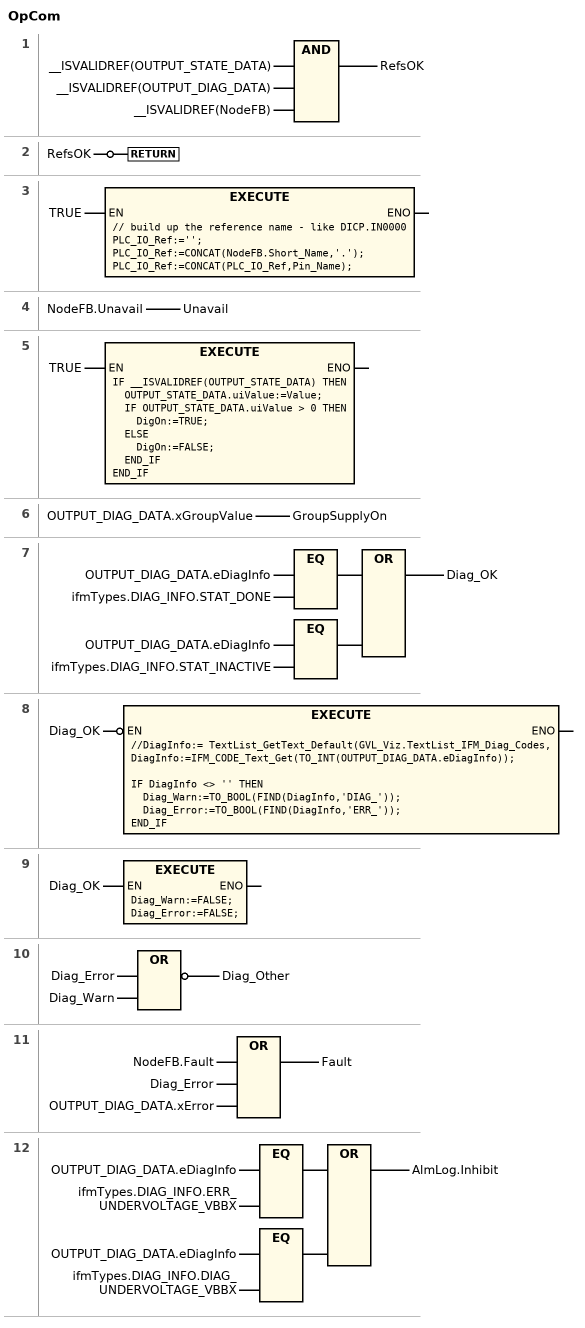
// NETWORK 1
RefsOK := (__ISVALIDREF(OUTPUT_STATE_DATA)) AND (__ISVALIDREF(OUTPUT_DIAG_DATA)) AND (__ISVALIDREF(NodeFB));

// NETWORK 2
IF NOT RefsOK THEN RETURN; END_IF

// NETWORK 3
// build up the reference name - like DICP.IN0000
PLC_IO_Ref:='';
PLC_IO_Ref:=CONCAT(NodeFB.Short_Name,'.');
PLC_IO_Ref:=CONCAT(PLC_IO_Ref,Pin_Name);

// NETWORK 4
Unavail := NodeFB.Unavail;

// NETWORK 5
IF __ISVALIDREF(OUTPUT_STATE_DATA) THEN
	OUTPUT_STATE_DATA.uiValue:=Value;
	IF OUTPUT_STATE_DATA.uiValue > 0 THEN
		DigOn:=TRUE;
	ELSE
		DigOn:=FALSE;
	END_IF
END_IF

// NETWORK 6
GroupSupplyOn := OUTPUT_DIAG_DATA.xGroupValue;

// NETWORK 7
Diag_OK := OUTPUT_DIAG_DATA.eDiagInfo = ifmTypes.DIAG_INFO.STAT_DONE OR OUTPUT_DIAG_DATA.eDiagInfo = ifmTypes.DIAG_INFO.STAT_INACTIVE;

// NETWORK 8
IF NOT Diag_OK THEN
    //DiagInfo:= TextList_GetText_Default(GVL_Viz.TextList_IFM_Diag_Codes,TO_STRING(OUTPUT_DIAG_DATA.eDiagInfo));
    DiagInfo:=IFM_CODE_Text_Get(TO_INT(OUTPUT_DIAG_DATA.eDiagInfo));
    
    IF DiagInfo <> '' THEN
    	Diag_Warn:=TO_BOOL(FIND(DiagInfo,'DIAG_'));	
    	Diag_Error:=TO_BOOL(FIND(DiagInfo,'ERR_'));	
    END_IF
END_IF

// NETWORK 9
IF Diag_OK THEN
    Diag_Warn:=FALSE;
    Diag_Error:=FALSE;
END_IF

// NETWORK 10
Diag_Other := NOT (Diag_Error OR Diag_Warn);

// NETWORK 11
Fault := NodeFB.Fault OR Diag_Error OR OUTPUT_DIAG_DATA.xError;

// NETWORK 12
AlmLog.Inhibit := OUTPUT_DIAG_DATA.eDiagInfo = ifmTypes.DIAG_INFO.ERR_UNDERVOLTAGE_VBBX OR OUTPUT_DIAG_DATA.eDiagInfo = ifmTypes.DIAG_INFO.DIAG_UNDERVOLTAGE_VBBX;

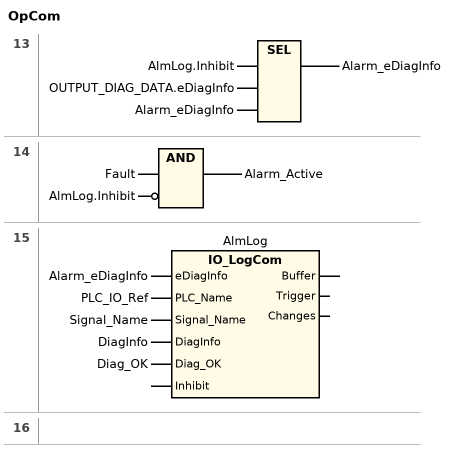
// NETWORK 13
Alarm_eDiagInfo := SEL(AlmLog.Inhibit, OUTPUT_DIAG_DATA.eDiagInfo, Alarm_eDiagInfo);

// NETWORK 14
Alarm_Active := Fault AND NOT AlmLog.Inhibit;

// NETWORK 15
AlmLog(
    eDiagInfo := Alarm_eDiagInfo,
    PLC_Name := PLC_IO_Ref,
    Signal_Name := Signal_Name,
    DiagInfo := DiagInfo,
    Diag_OK := Diag_OK); // IO_LogCom

// NETWORK 16

METHOD Init : BOOL
VAR_INPUT
	pPLC_Name: STRING;
	pSignal_Name: STRING;
	pPin_Name: STRING;
	pPin_Details: STRING;
	pOUTPUT_STATE_DATA: REFERENCE TO CRXXXX_OUTPUT_STATE_DATA;
	pOUTPUT_DIAG_DATA: REFERENCE TO CRXXXX_OUTPUT_DATA;
	pNodeFB: REFERENCE TO NodeComFB;	
END_VAR

PLC_Name:=pPLC_Name;
Signal_Name:=pSignal_Name;
Pin_Name:=pPin_Name;
Pin_Details:=pPin_Details;

OUTPUT_STATE_DATA REF= pOUTPUT_STATE_DATA;
OUTPUT_DIAG_DATA REF= pOUTPUT_DIAG_DATA;

NodeFB REF=pNodeFB;
END_METHOD

END_FUNCTION_BLOCK

// Device/Application/LIBS/IO Common/IFM_CODE_Text_Get
FUNCTION IFM_CODE_Text_Get : STRING
VAR_INPUT
	CODE: INT;
END_VAR
VAR
	TEXT: STRING;
END_VAR

IF CODE = 0 THEN
	TEXT:='STAT_INACTIVE';
END_IF;
IF CODE = 1 THEN
	TEXT:='STAT_DONE';
END_IF;
IF CODE = 2 THEN
	TEXT:='STAT_BUSY';
END_IF;
IF CODE = 3 THEN
	TEXT:='STAT_PREPARING';
END_IF;
IF CODE = 4 THEN
	TEXT:='STAT_READY';
END_IF;
IF CODE = 5 THEN
	TEXT:='STAT_RESET';
END_IF;
IF CODE = 6 THEN
	TEXT:='STAT_ABORTED';
END_IF;
IF CODE = 7 THEN
	TEXT:='RESERVED_07';
END_IF;
IF CODE = 8 THEN
	TEXT:='RESERVED_08';
END_IF;
IF CODE = 9 THEN
	TEXT:='RESERVED_09';
END_IF;
IF CODE = 10 THEN
	TEXT:='ERR_OPEN_CIRCUIT';
END_IF;
IF CODE = 11 THEN
	TEXT:='ERR_SHORT_CIRCUIT';
END_IF;
IF CODE = 12 THEN
	TEXT:='ERR_OVERLOAD_CURRENT';
END_IF;
IF CODE = 13 THEN
	TEXT:='ERR_LOW_CURRENT';
END_IF;
IF CODE = 14 THEN
	TEXT:='ERR_UNDERVOLTAGE_VBBX';
END_IF;
IF CODE = 15 THEN
	TEXT:='ERR_OVERVOLTAGE_VBBX';
END_IF;
IF CODE = 16 THEN
	TEXT:='ERR_STUCK_AT_HIGH';
END_IF;
IF CODE = 17 THEN
	TEXT:='ERR_STUCK_AT_LOW';
END_IF;
IF CODE = 18 THEN
	TEXT:='ERR_HIGH_TEMPERATURE';
END_IF;
IF CODE = 19 THEN
	TEXT:='ERR_LOW_TEMPERATURE';
END_IF;
IF CODE = 20 THEN
	TEXT:='ERR_INVALID_VALUE';
END_IF;
IF CODE = 21 THEN
	TEXT:='ERR_INVALID_CHANNEL';
END_IF;
IF CODE = 22 THEN
	TEXT:='ERR_INVALID_MODE';
END_IF;
IF CODE = 23 THEN
	TEXT:='ERR_INVALID_FREQUENCY';
END_IF;
IF CODE = 24 THEN
	TEXT:='ERR_INVALID_DITHER';
END_IF;
IF CODE = 25 THEN
	TEXT:='ERR_INVALID_FILTER';
END_IF;
IF CODE = 26 THEN
	TEXT:='ERR_UNREACHABLE_CURRENT';
END_IF;
IF CODE = 27 THEN
	TEXT:='ERR_SLOW_SIGNAL';
END_IF;
IF CODE = 28 THEN
	TEXT:='ERR_CHANGEOVER_TIME';
END_IF;
IF CODE = 29 THEN
	TEXT:='ERR_INSTANCE';
END_IF;
IF CODE = 30 THEN
	TEXT:='ERR_INSTANCE_LIMIT';
END_IF;
IF CODE = 31 THEN
	TEXT:='ERR_INVALID_COLOUR';
END_IF;
IF CODE = 32 THEN
	TEXT:='ERR_NO_IDENTITY';
END_IF;
IF CODE = 33 THEN
	TEXT:='ERR_ACCESS';
END_IF;
IF CODE = 34 THEN
	TEXT:='ERR_UNDEFINED';
END_IF;
IF CODE = 35 THEN
	TEXT:='ERR_FUNC_KEY_MISSED';
END_IF;
IF CODE = 36 THEN
	TEXT:='ERR_BUFFER_OVERFLOW';
END_IF;
IF CODE = 37 THEN
	TEXT:='ERR_BAUDRATE_ALREADY_SET';
END_IF;
IF CODE = 38 THEN
	TEXT:='ERR_INACTIVE_INTERFACE';
END_IF;
IF CODE = 39 THEN
	TEXT:='ERR_TIMEOUT';
END_IF;
IF CODE = 40 THEN
	TEXT:='ERR_OUT_OF_MEMORY';
END_IF;
IF CODE = 41 THEN
	TEXT:='ERR_BUS_OFF';
END_IF;
IF CODE = 42 THEN
	TEXT:='ERR_BAD_CRC';
END_IF;
IF CODE = 43 THEN
	TEXT:='ERR_EXCEEDED_RANGE';
END_IF;
IF CODE = 44 THEN
	TEXT:='ERR_INTERNAL_COMMUNICATION';
END_IF;
IF CODE = 45 THEN
	TEXT:='ERR_NOT_SUPPORTED';
END_IF;
IF CODE = 46 THEN
	TEXT:='ERR_TIMING';
END_IF;
IF CODE = 47 THEN
	TEXT:='ERR_INTERNAL';
END_IF;
IF CODE = 48 THEN
	TEXT:='ERR_FILE_SYSTEM';
END_IF;
IF CODE = 49 THEN
	TEXT:='ERR_INVALID_IP_CFG';
END_IF;
IF CODE = 50 THEN
	TEXT:='ERR_FAILED_ERR_RESET';
END_IF;
IF CODE = 51 THEN
	TEXT:='ERR_DEVICE_NOT_AVAILABLE';
END_IF;
IF CODE = 52 THEN
	TEXT:='ERR_NO_OBJECT';
END_IF;
IF CODE = 53 THEN
	TEXT:='ERR_UNREACHABLE_VOLTAGE';
END_IF;
IF CODE = 54 THEN
	TEXT:='ERR_AT_GROUP_OUTPUT';
END_IF;
IF CODE = 55 THEN
	TEXT:='ERR_CONTROL_DITHER';
END_IF;
IF CODE = 56 THEN
	TEXT:='ERR_UNDERVOLTAGE_VBBX_WARNING';
END_IF;
IF CODE = 57 THEN
	TEXT:='ERR_OVERVOLTAGE_VBBX_WARNING';
END_IF;
IF CODE = 58 THEN
	TEXT:='ERR_LOW_TEMPERATURE_WARNING';
END_IF;
IF CODE = 59 THEN
	TEXT:='ERR_HIGH_TEMPERATURE_WARNING';
END_IF;
IF CODE = 60 THEN
	TEXT:='ERR_RANGE_OVERRUN';
END_IF;
IF CODE = 61 THEN
	TEXT:='ERR_RANGE_UNDERRUN';
END_IF;
IF CODE = 62 THEN
	TEXT:='DIAG_INVALID_VALUE';
END_IF;
IF CODE = 63 THEN
	TEXT:='DIAG_INTERNAL';
END_IF;
IF CODE = 64 THEN
	TEXT:='DIAG_OPEN_CIRCUIT';
END_IF;
IF CODE = 65 THEN
	TEXT:='DIAG_SHORT_CIRCUIT';
END_IF;
IF CODE = 66 THEN
	TEXT:='DIAG_UNDERVOLTAGE_VBBX';
END_IF;
IF CODE = 67 THEN
	TEXT:='DIAG_OVERVOLTAGE_VBBX';
END_IF;
IF CODE = 68 THEN
	TEXT:='DIAG_OVERLOAD_CURRENT';
END_IF;
IF CODE = 69 THEN
	TEXT:='DIAG_STUCK_AT';
END_IF;
IF CODE = 70 THEN
	TEXT:='DIAG_STUCK_AT_HIGH';
END_IF;
IF CODE = 71 THEN
	TEXT:='DIAG_STUCK_AT_LOW';
END_IF;
IF CODE = 72 THEN
	TEXT:='DIAG_INVALID_COLOUR';
END_IF;
IF CODE = 73 THEN
	TEXT:='DIAG_OVERVOLTAGE';
END_IF;
IF CODE = 74 THEN
	TEXT:='DIAG_UNDERVOLTAGE';
END_IF;
IF CODE = 75 THEN
	TEXT:='DIAG_NO_CALIB';
END_IF;
IF CODE = 76 THEN
	TEXT:='DIAG_ACCESS';
END_IF;
IF CODE = 77 THEN
	TEXT:='DIAG_CHANGEOVER_TIME';
END_IF;
IF CODE = 78 THEN
	TEXT:='ERR_OVERVOLTAGE';
END_IF;
IF CODE = 79 THEN
	TEXT:='ERR_UNDERVOLTAGE';
END_IF;
IF CODE = 80 THEN
	TEXT:='ERR_STUCK_AT';
END_IF;
IF CODE = 81 THEN
	TEXT:='DIAG_CONTROL_DITHER';
END_IF;
IF CODE = 82 THEN
	TEXT:='DIAG_SLOW_SIGNAL';
END_IF;
IF CODE = 83 THEN
	TEXT:='DIAG_DIAG_PRO_MODE';
END_IF;
IF CODE = 84 THEN
	TEXT:='DIAG_WINDOW';
END_IF;
IF CODE = 85 THEN
	TEXT:='ERR_SDO_IDX_NOT_EXIST';
END_IF;
IF CODE = 86 THEN
	TEXT:='ERR_SDO_SUBIDX_NOT_EXIST';
END_IF;
IF CODE = 87 THEN
	TEXT:='ERR_SDO_UNSUPPORTED_ACCESS';
END_IF;
IF CODE = 88 THEN
	TEXT:='ERR_SDO_DATA_TYPE';
END_IF;
IF CODE = 89 THEN
	TEXT:='DIAG_LOW_TEMPERATURE';
END_IF;
IF CODE = 90 THEN
	TEXT:='DIAG_HIGH_TEMPERATURE';
END_IF;
IF CODE = 91 THEN
	TEXT:='DIAG_INVALID_DITHER';
END_IF;
IF CODE = 92 THEN
	TEXT:='DIAG_INVALID_FREQUENCY';
END_IF;
IF CODE = 93 THEN
	TEXT:='DIAG_RANGE_OVERRUN';
END_IF;
IF CODE = 94 THEN
	TEXT:='DIAG_RANGE_UNDERRUN';
END_IF;
IF CODE = 95 THEN
	TEXT:='DIAG_INVALID_FILTER';
END_IF;
IF CODE = 96 THEN
	TEXT:='ERR_COMPARE_MISMATCH';
END_IF;
IF CODE = 97 THEN
	TEXT:='DIAG_INVALID_IP_CFG';
END_IF;
IF CODE = 98 THEN
	TEXT:='DIAG_LOW_CURRENT';
END_IF;
IF CODE = 99 THEN
	TEXT:='DIAG_AT_GROUP_OUTPUT';
END_IF;
IF CODE = 100 THEN
	TEXT:='ERR_SDO_UNKNOWN';
END_IF;
IF CODE = 101 THEN
	TEXT:='ERR_BAUDRATE_INVALID_OR_ALREADY_SET';
END_IF;
IF CODE = 102 THEN
	TEXT:='DIAG_COMPARE_MISMATCH';
END_IF;
IF CODE = 103 THEN
	TEXT:='DIAG_COMPARE_MISMATCH_VSYS';
END_IF;
IF CODE = 104 THEN
	TEXT:='DIAG_GROUP_OVERLOAD_CURRENT';
END_IF;
IF CODE = 105 THEN
	TEXT:='ERR_GROUP_OVERLOAD_CURRENT';
END_IF;
IF CODE = 106 THEN
	TEXT:='STAT_PAUSED';
END_IF;
IF CODE = 107 THEN
	TEXT:='STAT_ABORT';
END_IF;
IF CODE = 108 THEN
	TEXT:='STAT_EVNT_OPEN_PLUG_STORAGE';
END_IF;
IF CODE = 109 THEN
	TEXT:='STAT_EVNT_OPEN_UNPLUG_STORAGE';
END_IF;
IF CODE = 110 THEN
	TEXT:='STAT_EVNT_OPEN_DONE';
END_IF;
IF CODE = 111 THEN
	TEXT:='STAT_EVNT_REGI_PLUG_STORAGE';
END_IF;
IF CODE = 112 THEN
	TEXT:='STAT_EVNT_REGI_UNPLUG_STORAGE';
END_IF;
IF CODE = 113 THEN
	TEXT:='STAT_EVNT_REGI_DONE';
END_IF;
IF CODE = 114 THEN
	TEXT:='STAT_EVNT_UNREGI';
END_IF;
IF CODE = 115 THEN
	TEXT:='STAT_EVNT_UNREGI_DONE';
END_IF;
IF CODE = 116 THEN
	TEXT:='STAT_EVNT_CLOSE';
END_IF;
IF CODE = 117 THEN
	TEXT:='STAT_EVNT_CLOSE_DONE';
END_IF;
IF CODE = 118 THEN
	TEXT:='ERR_INSTANCE_RESTRICTION';
END_IF;
IF CODE = 119 THEN
	TEXT:='ERR_NO_FILE';
END_IF;
IF CODE = 120 THEN
	TEXT:='ERR_EVNT_OPEN';
END_IF;
IF CODE = 121 THEN
	TEXT:='ERR_EVNT_REGI';
END_IF;
IF CODE = 122 THEN
	TEXT:='ERR_EVNT_UNREGI';
END_IF;
IF CODE = 123 THEN
	TEXT:='ERR_EVNT_CLOSE';
END_IF;
IF CODE = 124 THEN
	TEXT:='ERR_GET_STORAGE_LIST';
END_IF;
IF CODE = 125 THEN
	TEXT:='ERR_UNPLUG_STORAGE';
END_IF;
IF CODE = 126 THEN
	TEXT:='DIAG_INVALID_CHANNEL';
END_IF;
IF CODE = 127 THEN
	TEXT:='DIAG_INVALID_MODE';
END_IF;
IF CODE = 128 THEN
	TEXT:='ERR_H_BRIDGE_TEST';
END_IF;
IF CODE = 129 THEN
	TEXT:='ERR_GROUP_SW_TEST';
END_IF;
IF CODE = 130 THEN
	TEXT:='ERR_TX_ERROR';
END_IF;
IF CODE = 131 THEN
	TEXT:='ERR_RX_ERROR';
END_IF;
IF CODE = 132 THEN
	TEXT:='DIAG_PHASE_MISSING_B';
END_IF;
IF CODE = 133 THEN
	TEXT:='DIAG_PHASE_TOO_MANY_B';
END_IF;

IFM_CODE_Text_Get:=TEXT;

END_FUNCTION

// Device/Application/LIBS/IO Diagnostics/CRXXXX_Output_Display
FUNCTION_BLOCK CRXXXX_Output_Display
VAR_INPUT
	DisableMan:BOOL;
END_VAR
VAR_OUTPUT
	oPinDetailsStr:STRING;
	oSignalNameStr: STRING;
	oMainString: STRING; // could be Digital:ON/OFF, mV, mA or Hz PWM?
	oMainStringColour: DWORD;	
	oDiagStr: STRING; // Diagnostics info
	oShowDigRect:BOOL;
	oDigRectColour:DWORD;
	oTypeStr:STRING;
	oForceColour:DWORD;
	oForceText:STRING(5);
END_VAR
VAR
	InitDone:BOOL :=FALSE;	
	Update: BOOL:=TRUE;
	Update_Signal_Name: BOOL:=TRUE;	
	OpREF: REFERENCE TO OpCom;
	Pin_Name_Temp:STRING(10);
	Pin_Number_Temp:STRING(10);
	temp_real_mA:STRING(10);
	temp_real_mV:STRING(10);
	TextListItem:STRING;
	MainStringFlash: BOOL;
	UpdateDiag: BOOL;
	MainStringTemp: STRING;
END_VAR

VAR_IN_OUT
END_VAR

IF Update=FALSE THEN
	RETURN;
END_IF

IF __ISVALIDREF(OpREF) = FALSE THEN
	RETURN;
END_IF

IF OpREF.RefsOK = FALSE THEN
	RETURN;
END_IF

// set defaults first for the main string
oShowDigRect:=FALSE;
oTypeStr:='';
MainStringFlash:=FALSE;
oMainString:='';
MainStringTemp:='';
oMainStringColour:=GVL_Viz.Diag_Output_Font_Colour_OK;

// this code displays the Signal name - can be toggled using the function key
IF Update_Signal_Name THEN
	oPinDetailsStr:=OpREF.Pin_Name;
	IF GVL_Viz.Diag_Signal_Name_Toggle THEN
		TextListItem:=OpREF.Signal_Name;
		//oPinDetailsStr:=OpREF.Pin_Details;
	ELSE
		TextListItem:=Mimic_IO_GetText(GVL_Viz.TextList_IO_Diag,OpREF.PLC_IO_Ref);
		//oPinDetailsStr:=OpREF.Pin_Name;
	END_IF	
	
	IF (FIND(TextListItem,'Spare_') = 1) OR (FIND(TextListItem,'SPARE_') = 1) THEN
		// Starts with Spare
		oSignalNameStr:=' --- ';
	ELSE
		oSignalNameStr:=TextListItem;
	END_IF
END_IF

IF OpREF.Unavail THEN
	// the output is unvailable!
	IF GVL_Viz.Output_Fault_Flash_Slow THEN
		oMainString:=GVL_Viz.Diag_Output_Unavailable_Text;
		MainStringFlash:=TRUE;	
	END_IF
	oMainStringColour:=GVL_Viz.Diag_Output_Font_Colour_Unavail;
ELSIF OpREF.Diag_OK = FALSE THEN
	// something is not OK with the output
	// may be a fault or warning !
	IF GVL_Viz.Output_Fault_Flash_Slow THEN
		// do something if in this high period of the slow flash
		MainStringFlash:=TRUE;
		oMainString:=OpREF.DiagInfo;
	END_IF
	// always use the selected color - even if not showing the Diagnostic Info!
	IF OpREF.Diag_Error THEN
		oMainStringColour:=GVL_Viz.Diag_Output_Font_Colour_Error;
	ELSIF OpREF.Diag_Warn THEN
		oMainStringColour:=GVL_Viz.Diag_Output_Font_Colour_Warn;
	ELSE
		oMainStringColour:=GVL_Viz.Diag_Output_Font_Colour_Other;			
	END_IF			
END_IF

CASE OpREF.OUTPUT_DIAG_DATA.PWM_Flags OF		
Diag_Op_PWM_Enum.PWM_Single_Pin_CSO:		
	oTypeStr:='PWMH';
	UpdateDiag:=TRUE;
	
	MainStringTemp:= 'Act:';
	MainStringTemp:= TO_STRING(OpREF.OUTPUT_DIAG_DATA.uiOutCurrent);
	MainStringTemp:= CONCAT(MainStringTemp,'mA,');
	MainStringTemp:= CONCAT(MainStringTemp,'Trg:');
	MainStringTemp:= CONCAT(MainStringTemp,TO_STRING(OpREF.OUTPUT_DIAG_DATA.uiOpValue));
	MainStringTemp:= CONCAT(MainStringTemp,'mA');	
	
Diag_Op_PWM_Enum.PWM_Single_Pin_CSI:
	oTypeStr:='PWML';
	UpdateDiag:=TRUE;
Diag_Op_PWM_Enum.PWM_Bridge_A:
	oTypeStr:='PWMA';
	UpdateDiag:=TRUE;
Diag_Op_PWM_Enum.PWM_Bridge_B:
	oTypeStr:='PWMB';
	UpdateDiag:=TRUE;
END_CASE

CASE OpREF.OUTPUT_DIAG_DATA.eMode OF
ifmIOcommon.MODE_OUTPUT.OUT_DIGITAL_CSO:
	oShowDigRect:=TRUE;
	oTypeStr:='CSO-Hi';	
	UpdateDiag:=TRUE;
	temp_real_mV:=OSCAT_BASIC.REAL_TO_STRF(TO_REAL(OpREF.OUTPUT_DIAG_DATA.uiOutVoltage)/1000,2,'.');
	temp_real_mV:=CONCAT(temp_real_mV,'V');
	temp_real_mA:=OSCAT_BASIC.REAL_TO_STRF(TO_REAL(OpREF.OUTPUT_DIAG_DATA.uiOutCurrent)/1000,2,'.');
	temp_real_mA:=CONCAT(temp_real_mA,'A');
	
	MainStringTemp:= CONCAT(MainStringTemp,temp_real_mA);
	MainStringTemp:= CONCAT(MainStringTemp,',');
	
	MainStringTemp:= CONCAT(MainStringTemp,'Drv:');
	IF OpREF.OUTPUT_DIAG_DATA.xOutState = 0 THEN
		oDigRectColour:=GVL_Viz.IFM_IO_Output_DigRectColour_OFF;
		MainStringTemp:= CONCAT(MainStringTemp,'OFF');
	ELSE
		oDigRectColour:=GVL_Viz.IFM_IO_Output_DigRectColour_ON;
		MainStringTemp:= CONCAT(MainStringTemp,'ON');
	END_IF
	
	MainStringTemp:= CONCAT(MainStringTemp,',F.Back:');
	IF OpREF.OUTPUT_DIAG_DATA.uiOpValue = 0 THEN
		MainStringTemp:= CONCAT(MainStringTemp,'OFF');
	ELSE
		MainStringTemp:= CONCAT(MainStringTemp,'ON');
	END_IF	

ifmIOcommon.MODE_OUTPUT.OUT_ANALOGUE_10:
	oShowDigRect:=TRUE;
	oTypeStr:='An_10v';
	UpdateDiag:=TRUE;
			
	temp_real_mV:=OSCAT_BASIC.REAL_TO_STRF(TO_REAL(OpREF.OUTPUT_DIAG_DATA.uiOutVoltage)/1000,2,'.');
	temp_real_mV:=CONCAT(temp_real_mV,'V');
	temp_real_mA:=TO_STRING(OpREF.OUTPUT_DIAG_DATA.uiOutCurrent);
	temp_real_mA:=CONCAT(temp_real_mA,'mA');
	
	MainStringTemp:= '';
	MainStringTemp:= CONCAT(MainStringTemp,temp_real_mV);
	MainStringTemp:= CONCAT(MainStringTemp,',');
	MainStringTemp:= CONCAT(MainStringTemp,temp_real_mA);
	MainStringTemp:= CONCAT(MainStringTemp,',');
	
	IF OpREF.OUTPUT_DIAG_DATA.xOutState = TRUE THEN
		oDigRectColour:=GVL_Viz.IFM_IO_Output_DigRectColour_ON;
		MainStringTemp:= CONCAT(MainStringTemp,'ON');
	ELSE
		oDigRectColour:=GVL_Viz.IFM_IO_Output_DigRectColour_OFF;
		MainStringTemp:= CONCAT(MainStringTemp,'OFF');
	END_IF
	
	MainStringTemp:= CONCAT(MainStringTemp,',D:');
	MainStringTemp:= CONCAT(MainStringTemp,TO_STRING(OpREF.OUTPUT_DIAG_DATA.uiOpValue));
	
ifmIOcommon.MODE_OUTPUT.OUT_SENSOR_10,
ifmIOcommon.MODE_OUTPUT.OUT_SENSOR_05:
	oShowDigRect:=TRUE;
	IF OpREF.OUTPUT_DIAG_DATA.eMode = ifmIOcommon.MODE_OUTPUT.OUT_SENSOR_05 THEN
		oTypeStr:='5v_Sup';
	ELSE
		oTypeStr:='10v_Sup';
	END_IF
	UpdateDiag:=TRUE;
	
	temp_real_mV:=OSCAT_BASIC.REAL_TO_STRF(TO_REAL(OpREF.OUTPUT_DIAG_DATA.uiOutVoltage)/1000,2,'.');
	temp_real_mV:=CONCAT(temp_real_mV,'V');
	temp_real_mA:=TO_STRING(OpREF.OUTPUT_DIAG_DATA.uiOutCurrent);
	temp_real_mA:=CONCAT(temp_real_mA,'mA');
	
	MainStringTemp:= '';
	MainStringTemp:= CONCAT(MainStringTemp,temp_real_mV);
	MainStringTemp:= CONCAT(MainStringTemp,',');
	MainStringTemp:= CONCAT(MainStringTemp,temp_real_mA);
	MainStringTemp:= CONCAT(MainStringTemp,',');
	
	IF OpREF.OUTPUT_DIAG_DATA.xOutState = TRUE THEN
		oDigRectColour:=GVL_Viz.IFM_IO_Output_DigRectColour_ON;
		MainStringTemp:= CONCAT(MainStringTemp,'ON');
	ELSE
		oDigRectColour:=GVL_Viz.IFM_IO_Output_DigRectColour_OFF;
		MainStringTemp:= CONCAT(MainStringTemp,'OFF');
	END_IF
	
	MainStringTemp:= CONCAT(MainStringTemp,',D:');
	MainStringTemp:= CONCAT(MainStringTemp,TO_STRING(OpREF.OUTPUT_DIAG_DATA.uiOpValue));
END_CASE
	
IF MainStringFlash = FALSE THEN
	oMainString:=MainStringTemp;
END_IF

// this is the basic text box to the right - uses same colour as the main string
IF OpREF.Diag_OK THEN
	oDiagStr:='Diag:OK';
ELSE
	IF OpREF.Diag_Error = TRUE THEN
		oDiagStr:='Err.:';
	ELSIF OpREF.Diag_Warn = TRUE THEN
		oDiagStr:='Warn:';
	ELSE
		oDiagStr:='Oth:';
	END_IF
	oDiagStr:=CONCAT(oDiagStr,TO_STRING(OpREF.OUTPUT_DIAG_DATA.eDiagInfo));
END_IF

// add the optional diagnostic string - maybe scaling information 
IF 	UpdateDiag=TRUE THEN
	IF LEN(OpREF.DiagString) > 0 THEN
		IF LEN(oMainString) > 0 THEN
			oMainString:= CONCAT(oMainString,',');		
		END_IF
		oMainString:= CONCAT(oMainString,OpREF.DiagString);
	END_IF	
END_IF

// show a special colour and M is the output is being force on with PLC Manual.
IF OpREF.OUTPUT_STATE_DATA.xManAuto THEN
	oForceText:='M';
	IF OpREF.OUTPUT_STATE_DATA.uiManValue > 0 THEN
		oForceColour:=GVL_Viz.IFM_IO_Output_DigRectColour_ManOn;
	ELSE
		oForceColour:=GVL_Viz.IFM_IO_Output_DigRectColour_ManOff;
	END_IF
ELSE
	oForceText:='';
	oForceColour:=16#FFFFFFFF;
END_IF

METHOD Init : BOOL
VAR_INPUT
	pOpREF: REFERENCE TO OpCom;
END_VAR
OpREF REF= pOpREF;
InitDone:=TRUE;
END_METHOD

END_FUNCTION_BLOCK

// Project Information/GetCompany
// This function has been automatically generated from the project information.
{attribute 'signature_flag' := '1073741824'}
{attribute 'register_in_runtime'}
FUNCTION GetCompany : WSTRING
VAR_INPUT
	
END_VAR

GetCompany := "MTech";

END_FUNCTION

// Project Information/GetTitle
// This function has been automatically generated from the project information.
{attribute 'signature_flag' := '1073741824'}
{attribute 'register_in_runtime'}
FUNCTION GetTitle : WSTRING
VAR_INPUT
	
END_VAR

GetTitle := "MAIN_HMI";

END_FUNCTION

// Project Information/GetVersion
// This function has been automatically generated from the project information.
{attribute 'signature_flag' := '1073741824'}
{attribute 'register_in_runtime'}
FUNCTION GetVersion : VERSION
VAR_INPUT
	
END_VAR

GetVersion.uiMajor := 3;
GetVersion.uiMinor := 0;
GetVersion.uiServicePack := 0;
GetVersion.uiPatch := 7;

END_FUNCTION

// Project Information/GetTextProperty
// This function has been automatically generated from the project information.
{attribute 'signature_flag' := '1073741824'}
{attribute 'register_in_runtime'}
FUNCTION GetTextProperty : WSTRING
VAR_INPUT
	stKey: WSTRING;
END_VAR

IF stKey = "Author" THEN
	GetTextProperty := "AW";
ELSIF stKey = "Company" THEN
	GetTextProperty := "MTech";
ELSIF stKey = "CompileDateTime" THEN
	GetTextProperty := "09:01:42,04-04-2025";
ELSIF stKey = "DefaultNamespace" THEN
	GetTextProperty := "";
ELSIF stKey = "Description" THEN
	GetTextProperty := "T620X/Radial";
ELSIF stKey = "Project" THEN
	GetTextProperty := "T620X_HMI_CR1076_SP19p4";
ELSIF stKey = "Title" THEN
	GetTextProperty := "MAIN_HMI";
ELSE
	GetTextProperty := "";
END_IF

END_FUNCTION

// Project Information/GetTextProperty2
// This function has been automatically generated from the project information.
{attribute 'signature_flag' := '1073741824'}
{attribute 'register_in_runtime'}
FUNCTION GetTextProperty2 : POINTER TO WSTRING
VAR_INPUT
	stKey: WSTRING;
END_VAR

IF stKey = "Author" THEN
	GetTextProperty2 := ADR("AW");
ELSIF stKey = "Company" THEN
	GetTextProperty2 := ADR("MTech");
ELSIF stKey = "CompileDateTime" THEN
	GetTextProperty2 := ADR("09:01:42,04-04-2025");
ELSIF stKey = "DefaultNamespace" THEN
	GetTextProperty2 := ADR("");
ELSIF stKey = "Description" THEN
	GetTextProperty2 := ADR("T620X/Radial");
ELSIF stKey = "Project" THEN
	GetTextProperty2 := ADR("T620X_HMI_CR1076_SP19p4");
ELSIF stKey = "Title" THEN
	GetTextProperty2 := ADR("MAIN_HMI");
ELSE
	GetTextProperty2 := ADR("");
END_IF

END_FUNCTION

// Project Information/GetNumberProperty
// This function has been automatically generated from the project information.
{attribute 'signature_flag' := '1073741824'}
{attribute 'register_in_runtime'}
FUNCTION GetNumberProperty : DINT
VAR_INPUT
	stKey: WSTRING;
END_VAR

GetNumberProperty := 0;

END_FUNCTION

// Project Information/GetBooleanProperty
// This function has been automatically generated from the project information.
{attribute 'signature_flag' := '1073741824'}
{attribute 'register_in_runtime'}
FUNCTION GetBooleanProperty : BOOL
VAR_INPUT
	stKey: WSTRING;
END_VAR

IF stKey = "Released" THEN
	GetBooleanProperty := FALSE;
ELSE
	GetBooleanProperty := FALSE;
END_IF

END_FUNCTION

// Project Information/GetVersionProperty
// This function has been automatically generated from the project information.
{attribute 'signature_flag' := '1073741824'}
{attribute 'register_in_runtime'}
FUNCTION GetVersionProperty : VERSION
VAR_INPUT
	stKey: WSTRING;
END_VAR

IF stKey = "Version" THEN
	GetVersionProperty.uiMajor := 3;
	GetVersionProperty.uiMinor := 0;
	GetVersionProperty.uiServicePack := 0;
	GetVersionProperty.uiPatch := 7;
ELSE
	GetVersionProperty.uiMajor := 0;
	GetVersionProperty.uiMinor := 0;
	GetVersionProperty.uiServicePack := 0;
	GetVersionProperty.uiPatch := 0;
END_IF

END_FUNCTION

// Device/Application/LIBS/IO Diagnostics/Diag_Ip_Freq_Pulse_FB
FUNCTION_BLOCK Diag_Ip_Freq_Pulse_FB
VAR_INPUT
	FormatString: STRING:='%.1fHz';
	Freq:REAL;
	Pulse:UDINT;	
END_VAR
VAR_OUTPUT
	OpString: STRING;
END_VAR
VAR
	TempString: STRING;
	Sprintf_Result: INT;
	
	Pointer_Test: POINTER TO IpCom;
	CAS_DriveShaftRpm_Diag_String: STRING;	
END_VAR

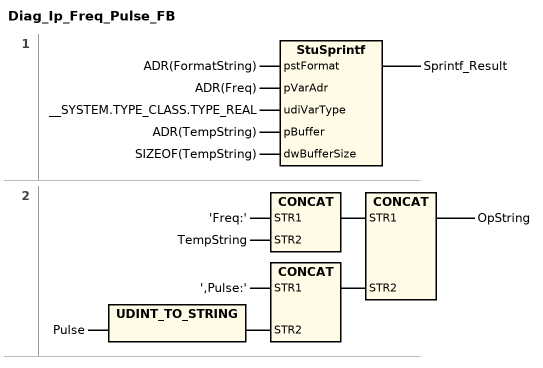
// NETWORK 1
Sprintf_Result := StuSprintf(pstFormat := ADR(FormatString), pVarAdr := ADR(Freq), udiVarType := __SYSTEM.TYPE_CLASS.TYPE_REAL, pBuffer := ADR(TempString), dwBufferSize := SIZEOF(TempString));

// NETWORK 2
OpString := CONCAT(STR1 := CONCAT(STR1 := 'Freq:', STR2 := TempString), STR2 := CONCAT(STR1 := ',Pulse:', STR2 := UDINT_TO_STRING(Pulse)));

END_FUNCTION_BLOCK

// Device/Application/LIBS/IO Diagnostics/CRXXXX_Output_Group_Display
FUNCTION_BLOCK CRXXXX_Output_Group_Display
VAR_INPUT
END_VAR
VAR_OUTPUT
	oPinDetailsStr:STRING;
	oSignalNameStr: STRING;
	oMainString: STRING; // could be Digital:ON/OFF, mV, mA or Hz PWM?
	oMainStringColour: DWORD;
//	oMainStringFillColour: DWORD;
	oDiagStr: STRING; // Diagnostics info
	oShowDigRect:BOOL;
	oDigRectColour:DWORD;
	oTypeStr:STRING;
	oDiagRectColour:DWORD;
END_VAR
VAR
	InitDone:BOOL :=FALSE;
	Update: BOOL:=TRUE;
	OpGrpREF: REFERENCE TO OpGrpCom;
	Pin_Name_Temp:STRING(10);
	Pin_Number_Temp:STRING(10);
	temp_real_mA:STRING(10);
	temp_real_mV:STRING(10);
	TextListItem:STRING;
	INIT_LABELS:BOOL:=TRUE;
	MainStringFlash:BOOL;
	PLC_IO_Ref:STRING;		
END_VAR

IF Update=FALSE THEN
	RETURN;
END_IF

IF __ISVALIDREF(OpGrpREF) = FALSE THEN
	RETURN;
END_IF

IF OpGrpREF.RefsOK = FALSE THEN
	RETURN;
END_IF

// build up the reference name - like DICP.IN0000
PLC_IO_Ref:='';
PLC_IO_Ref:=CONCAT(OpGrpRef.NodeFB.Short_Name,'.');
PLC_IO_Ref:=CONCAT(PLC_IO_Ref,OpGrpREF.Pin_Name);

IF INIT_LABELS THEN	
	oPinDetailsStr:=OpGrpREF.Pin_Name;
	IF GVL_Viz.Diag_Signal_Name_Toggle THEN
		TextListItem:=OpGrpREF.Signal_Name;
		//oPinDetailsStr:=OpGrpREF.Pin_Details;		
	ELSE
		//oPinDetailsStr:=OpGrpREF.Pin_Name;
		TextListItem:=Mimic_IO_GetText(GVL_Viz.TextList_IO_Mimics_Outputs,OpGrpREF.Signal_Name);
	END_IF	
	
	IF LEN(TextListItem)>0 THEN
		// we have some pin details - stop updating!
		//INIT_LABELS:=FALSE;
	END_IF;
	
	IF (FIND(TextListItem,'Spare_') = 1) OR (FIND(TextListItem,'SPARE_') = 1) THEN
		// Starts with Spare
		oSignalNameStr:=' --- ';
	ELSE
		oSignalNameStr:=TextListItem;
	END_IF	
END_IF

oShowDigRect:=TRUE;
oTypeStr:='Supply';

// set defaults first for the main string
MainStringFlash:=FALSE;
oMainString:='';
oMainStringColour:=GVL_Viz.Diag_Output_Font_Colour_OK;

IF OpGrpREF.Unavail THEN
	IF GVL_Viz.Output_Fault_Flash_Slow THEN
		oMainString:=GVL_Viz.Diag_Output_Unavailable_Text;
		MainStringFlash:=TRUE;		
	END_IF
	oMainStringColour:=GVL_Viz.Diag_Output_Font_Colour_Unavail;
END_IF

IF OpGrpREF.Fault THEN
	IF GVL_Viz.Output_Fault_Flash_Slow THEN
		MainStringFlash:=TRUE;
		//oMainString:=GVL_Viz.Diag_Output_Group_Fault_Text;
		oMainString:=Mimic_IO_GetText(GVL_Viz.TextList_IFM_Diag_Codes,TO_STRING(OpGrpREF.OUTPUT_GROUP_DIAG_DATA.eDiagInfo));;
	END_IF
	oMainStringColour:=GVL_Viz.Diag_Output_Font_Colour_Error;
END_IF

IF MainStringFlash = FALSE THEN
	temp_real_mV:=OSCAT_BASIC.REAL_TO_STRF(TO_REAL(OpGrpREF.OUTPUT_GROUP_DIAG_DATA.uiGroupVoltage)/1000,2,'.');
	temp_real_mV:=CONCAT(temp_real_mV,'V');
	temp_real_mA:=OSCAT_BASIC.REAL_TO_STRF(TO_REAL(OpGrpREF.OUTPUT_GROUP_DIAG_DATA.uiGroupCurrent)/1000,2,'.');
	temp_real_mA:=CONCAT(temp_real_mA,'A');
	
	oMainString:= CONCAT(oMainString,temp_real_mV);
	oMainString:= CONCAT(oMainString,',');
	oMainString:= CONCAT(oMainString,temp_real_mA);
	oMainString:= CONCAT(oMainString,',');
	
	IF OpGrpREF.OUTPUT_GROUP_DIAG_DATA.xGroupState = TRUE THEN
		oDigRectColour:=GVL_Viz.IFM_IO_Output_DigRectColour_ON;
		oMainString:= CONCAT(oMainString,'ON');
	ELSE
		oDigRectColour:=GVL_Viz.IFM_IO_Output_DigRectColour_OFF;
		oMainString:= CONCAT(oMainString,'OFF');
	END_IF
	
	oMainString:= CONCAT(oMainString,',in:');
	temp_real_mV:=OSCAT_BASIC.REAL_TO_STRF(TO_REAL(OpGrpREF.OUTPUT_GROUP_DIAG_DATA.uiVBBxVoltage)/1000,2,'.');
	temp_real_mV:=CONCAT(temp_real_mV,'V');	
	oMainString:= CONCAT(oMainString,temp_real_mV);	
END_IF

IF OpGrpREF.OUTPUT_GROUP_DIAG_DATA.eDiagInfo = ifmTypes.DIAG_INFO.STAT_DONE THEN
	oDiagStr:='Diag:OK';
ELSE
	IF OpGrpREF.OUTPUT_GROUP_DIAG_DATA.xError = TRUE THEN
		oDiagStr:='Err.:';
	ELSE	
		oDiagStr:='Diag:';
	END_IF	
	oDiagStr:=CONCAT(oDiagStr,TO_STRING(OpGrpREF.OUTPUT_GROUP_DIAG_DATA.eDiagInfo));
END_IF

METHOD Init : BOOL
VAR_INPUT
	pOpGrpREF: REFERENCE TO OpGrpCom;
END_VAR
OpGrpREF REF= pOpGrpREF;
InitDone:=TRUE;
END_METHOD

END_FUNCTION_BLOCK

// Device/Application/LIBS/IO Common/OpGrpCom
FUNCTION_BLOCK OpGrpCom

VAR_INPUT
END_VAR

VAR
	OUTPUT_STATE_DATA: REFERENCE TO CRXXXX_OUTPUT_STATE_DATA;
	OUTPUT_GROUP_DIAG_DATA: REFERENCE TO CRXXXX_OUTPUT_GROUP_DATA;

	PLC_Name: STRING;
	Signal_Name: STRING;
	Pin_Name: STRING;
	Pin_Details: STRING;
	
	NodeFB: REFERENCE TO NodeComFB;	

	RefsOK: BOOL;

	Diag_OK:BOOL;
	Diag_Error:BOOL;
	Diag_Warn:BOOL;
	Diag_Other:BOOL;
	
	Fault:BOOL;
	Unavail:BOOL;
	
	DiagInfo:STRING:='';
	PLC_IO_Ref:STRING;
	
	Alarm_eDiagInfo:ifmTypes.DIAG_INFO;		
	AlmLog: IO_LogCom;
	Alarm_Active: BOOL;		
END_VAR

VAR_OUTPUT
END_VAR

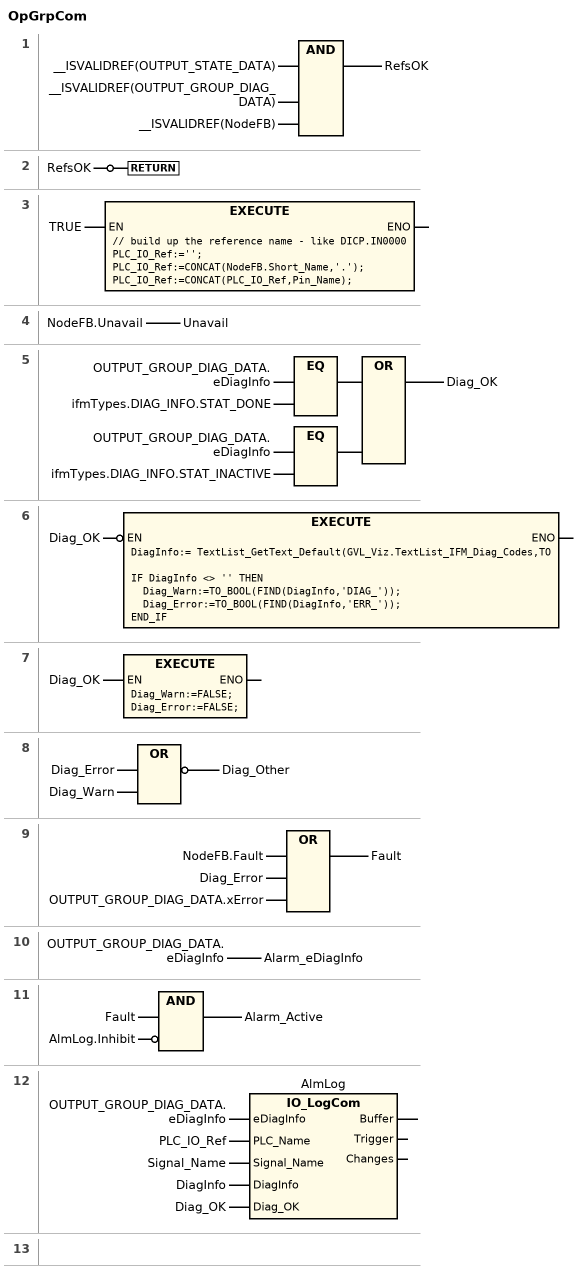
// NETWORK 1
RefsOK := (__ISVALIDREF(OUTPUT_STATE_DATA)) AND (__ISVALIDREF(OUTPUT_GROUP_DIAG_DATA)) AND (__ISVALIDREF(NodeFB));

// NETWORK 2
IF NOT RefsOK THEN RETURN; END_IF

// NETWORK 3
// build up the reference name - like DICP.IN0000
PLC_IO_Ref:='';
PLC_IO_Ref:=CONCAT(NodeFB.Short_Name,'.');
PLC_IO_Ref:=CONCAT(PLC_IO_Ref,Pin_Name);

// NETWORK 4
Unavail := NodeFB.Unavail;

// NETWORK 5
Diag_OK := OUTPUT_GROUP_DIAG_DATA.eDiagInfo = ifmTypes.DIAG_INFO.STAT_DONE OR OUTPUT_GROUP_DIAG_DATA.eDiagInfo = ifmTypes.DIAG_INFO.STAT_INACTIVE;

// NETWORK 6
IF NOT Diag_OK THEN
    DiagInfo:= TextList_GetText_Default(GVL_Viz.TextList_IFM_Diag_Codes,TO_STRING(OUTPUT_GROUP_DIAG_DATA.eDiagInfo));
    
    IF DiagInfo <> '' THEN
    	Diag_Warn:=TO_BOOL(FIND(DiagInfo,'DIAG_'));	
    	Diag_Error:=TO_BOOL(FIND(DiagInfo,'ERR_'));	
    END_IF
END_IF

// NETWORK 7
IF Diag_OK THEN
    Diag_Warn:=FALSE;
    Diag_Error:=FALSE;
END_IF

// NETWORK 8
Diag_Other := NOT (Diag_Error OR Diag_Warn);

// NETWORK 9
Fault := NodeFB.Fault OR Diag_Error OR OUTPUT_GROUP_DIAG_DATA.xError;

// NETWORK 10
Alarm_eDiagInfo := OUTPUT_GROUP_DIAG_DATA.eDiagInfo;

// NETWORK 11
Alarm_Active := Fault AND NOT AlmLog.Inhibit;

// NETWORK 12
AlmLog(
    eDiagInfo := OUTPUT_GROUP_DIAG_DATA.eDiagInfo,
    PLC_Name := PLC_IO_Ref,
    Signal_Name := Signal_Name,
    DiagInfo := DiagInfo,
    Diag_OK := Diag_OK); // IO_LogCom

// NETWORK 13

PROPERTY Dig : BOOL
GET
IF __ISVALIDREF(OUTPUT_STATE_DATA) THEN
	Dig:=TO_BOOL(OUTPUT_STATE_DATA.uiValue);
END_IF
END_GET
SET
VAR
	SET_UPDATES: DWORD;
END_VAR
IF __ISVALIDREF(OUTPUT_STATE_DATA) THEN
	OUTPUT_STATE_DATA.uiValue:=TO_UINT(Dig);
	SET_UPDATES:=SET_UPDATES+1;
END_IF
END_SET
END_PROPERTY

METHOD Init : BOOL
VAR_INPUT
	pPLC_Name: STRING;
	pSignal_Name: STRING;
	pPin_Name: STRING;
	pPin_Details: STRING;
	pOUTPUT_STATE_DATA: REFERENCE TO CRXXXX_OUTPUT_STATE_DATA;
	pOUTPUT_GROUP_DIAG_DATA: REFERENCE TO CRXXXX_OUTPUT_GROUP_DATA;
	pNodeFB: REFERENCE TO NodeComFB;	
END_VAR

PLC_Name:=pPLC_Name;
Signal_Name:=pSignal_Name;
Pin_Name:=pPin_Name;
Pin_Details:=pPin_Details;

OUTPUT_STATE_DATA REF= pOUTPUT_STATE_DATA;
OUTPUT_GROUP_DIAG_DATA REF= pOUTPUT_GROUP_DIAG_DATA;

NodeFB REF=pNodeFB;
END_METHOD

END_FUNCTION_BLOCK

// Device/Application/LIBS/Alarms/Functions/Alarm_Log_File_Write
FUNCTION Alarm_Log_File_Write : INT
VAR_INPUT
	LIST: REFERENCE TO SLL_LOGGER_MAIN_SRUCT;	
	szFileName : STRING:='AlarmBuffer.bin';	
	UpdatedCount: REFERENCE TO INT;
END_VAR
VAR	
	ReturnValue: INT:=-1;
	hFile : RTS_IEC_HANDLE := RTS_INVALID_HANDLE;
	
	udiWriteError : RTS_IEC_RESULT;
	udiOpenError : RTS_IEC_RESULT;
	udiCloseError : RTS_IEC_RESULT;
	udiWrite : __XWORD;
END_VAR

hFile := SysFileOpen(szFile:=szFileName, am:=SysFile.AM_APPEND_PLUS, pResult:=ADR(udiOpenError));

IF hFile <> RTS_INVALID_HANDLE	THEN
	udiWrite := SysFileWrite(hFile:=hFile, pbyBuffer:=ADR(LIST),ulSize:=TO_UDINT(LIST), pResult:=ADR(udiWriteError));
	udiCloseError  := SysFileClose(hFile:=hFile);
	Log_File_Append:=0;
	UpdatedCount:=UpdatedCount+1;
	RETURN;
END_IF

Alarm_Log_File_Write := ReturnValue;
RETURN;

END_FUNCTION

// Device/Application/LIBS/Alarms/Functions/Alarm_Log_Count_Active_Hush
FUNCTION Alarm_Log_Count_Active_Hush : INT

VAR_INPUT
	LIST: REFERENCE TO SLL_LOGGER_MAIN_SRUCT;
END_VAR
VAR_OUTPUT
	Hush_ActiveCount:INT:=0;
	Hush_InActiveCount:INT:=0;
END_VAR
VAR
	ErrorApp_Count:INT:=0;
	ErrorIO_Count:INT:=0;
	X:WORD;
END_VAR

ErrorApp_Count:=0;
ErrorIO_Count:=0;

Hush_ActiveCount:=0;
Hush_InActiveCount:=0;

FOR X :=0 TO (LIST.LOGGER_LIST_SIZE-1) BY 1 DO
	IF LIST.LOGGER_LIST[X].Group.ErrorApp THEN
		
		IF LIST.LOGGER_LIST[X].Group.HushOption = FALSE THEN
			// Normal Alarm - no Hush
			IF LIST.LOGGER_LIST[X].Flags.Active THEN
				ErrorApp_Count:=ErrorApp_Count+1;
			END_IF
		ELSE
			// Hush alarm option!			
			IF LIST.LOGGER_LIST[X].Flags.Active THEN
				Hush_ActiveCount:=Hush_ActiveCount+1;
			ELSE
				Hush_InActiveCount:=Hush_InActiveCount+1;
			END_IF
		END_IF
		
	END_IF
	IF LIST.LOGGER_LIST[X].Group.ErrorIO THEN
		ErrorIO_Count:=ErrorIO_Count+1;
	END_IF
END_FOR

Alarm_Log_Count_Active_Hush:=ErrorApp_Count+ErrorIO_Count+Hush_ActiveCount;

END_FUNCTION

// Device/Application/LIBS/Convert_mm_to_in_ft
FUNCTION_BLOCK Convert_mm_to_in_ft
VAR_INPUT
	mm_in: REAL;
	inches_format: STRING:='%.01fin.';
	feet_format: STRING:='%dft.';
END_VAR
VAR_OUTPUT
	Total_Inches: REAL;
	Feet: INT;
	Inches: REAL;
	Str:STRING;
END_VAR
VAR
	temp_inches_real: REAL;
//	temp_inches_int: INT;
	temp_ft_in_str: STRING;
	div_FEET: INT;
	mod_INCHES: REAL;
	fp_factor:INT :=100;
END_VAR

temp_ft_in_str:='';

temp_inches_real := TO_REAL(mm_in) / 25.4;
//temp_inches_int := TO_INT(temp_inches_real);

mod_INCHES:= OSCAT_BASIC.MODR(temp_inches_real,12);
div_FEET  := TO_INT(temp_inches_real/12);

Total_Inches:= (div_FEET * 12) + mod_INCHES;

IF div_FEET > 0 THEN
	temp_ft_in_str := print_formated_REAl_func('',feet_format,div_FEET);
END_IF

//IF mod_INCHES > 0 THEN	
	temp_ft_in_str := CONCAT(temp_ft_in_str,print_formated_REAl_func(' ',inches_format,mod_INCHES));
//END_IF

//IF div_FEET = 0 AND mod_INCHES = 0 THEN
//	temp_ft_in_str:= '0 in.';
//END_IF

Str:=temp_ft_in_str;
Inches:=mod_INCHES;
Feet:=div_FEET;

END_FUNCTION_BLOCK

// Device/Application/LIBS/print_formated_REAL_func
FUNCTION print_formated_REAL_func : STRING
VAR_INPUT
	Prefix: STRING;
	FormatString: STRING:='%0.1f';
	Value:REAL;	
END_VAR
VAR
	TempString: STRING;
END_VAR

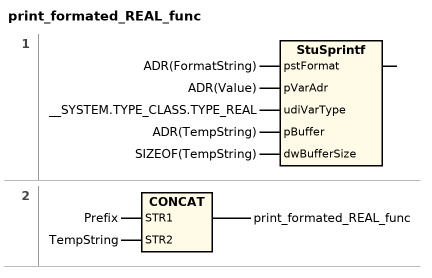
// NETWORK 1
StuSprintf(pstFormat := ADR(FormatString), pVarAdr := ADR(Value), udiVarType := __SYSTEM.TYPE_CLASS.TYPE_REAL, pBuffer := ADR(TempString), dwBufferSize := SIZEOF(TempString));

// NETWORK 2
print_formated_REAL_func := CONCAT(STR1 := Prefix, STR2 := TempString);

END_FUNCTION

// Device/Application/LIBS/SIMPLE_HB_CHECK_ONLINE
FUNCTION_BLOCK SIMPLE_HB_CHECK_ONLINE
VAR_INPUT
	TICKMS_IN: DWORD;
	ONLINE_TM: TIME:=T#500MS;
	OFFLINE_TM: TIME:=T#500MS;
END_VAR
VAR_OUTPUT
	ONLINE: BOOL;
END_VAR
VAR
	ONLINE_TON: TON;
	OFFLINE_TON: TON;
	TICKMS_PREV: DWORD;
END_VAR

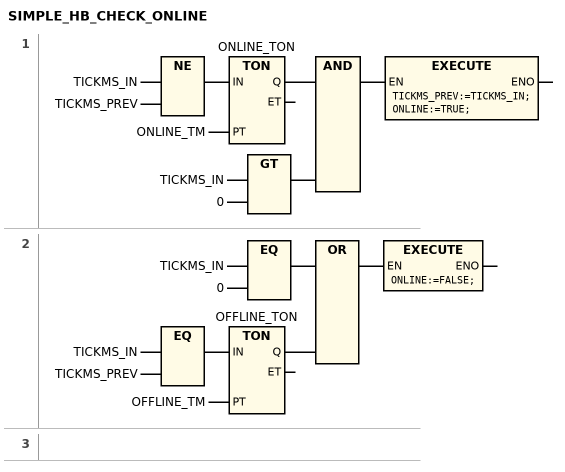
// NETWORK 1
ONLINE_TON(IN := TICKMS_IN <> TICKMS_PREV, PT := ONLINE_TM); // TON
IF ONLINE_TON.Q AND TICKMS_IN > 0 THEN
    TICKMS_PREV:=TICKMS_IN;
    ONLINE:=TRUE;
END_IF

// NETWORK 2
OFFLINE_TON(IN := TICKMS_IN = TICKMS_PREV, PT := OFFLINE_TM); // TON
IF TICKMS_IN = 0 OR OFFLINE_TON.Q THEN ONLINE:=FALSE; END_IF

// NETWORK 3

END_FUNCTION_BLOCK

// Device/Application/LIBS/print_BOOL_func
FUNCTION print_BOOL_func : STRING
VAR_INPUT
	Prefix: STRING;
	Value:BOOL;	
END_VAR
VAR
	TempString: STRING;
END_VAR

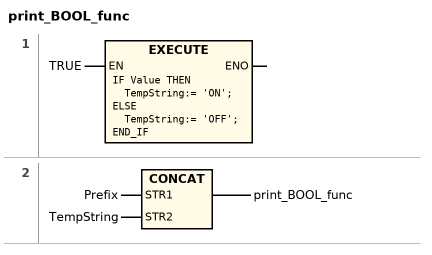
// NETWORK 1
IF Value THEN
	TempString:= 'ON';
ELSE
	TempString:= 'OFF';	
END_IF

// NETWORK 2
print_BOOL_func := CONCAT(STR1 := Prefix, STR2 := TempString);

END_FUNCTION

// Device/Application/LIBS/Alarms/Functions/Alarm_Log_Count_Errors_Hush
PROGRAM Alarm_Log_Count_Errors_Hush
VAR
END_VAR

// NETWORK 1

END_PROGRAM

// Device/Application/LIBS/Convert_inches_to_in_ft
FUNCTION_BLOCK Convert_inches_to_in_ft
VAR_INPUT
	inches_in: REAL;
	inches_format: STRING:='%.01fin.';
	feet_format: STRING:='%dft.';
END_VAR
VAR_OUTPUT
	Total_Inches: REAL;
	Feet: INT;
	Inches: REAL;
	Str:STRING;
END_VAR
VAR
	temp_ft_in_str: STRING;
	div_FEET: REAL;
	mod_INCHES: REAL;
	fp_factor:INT :=100;
END_VAR

temp_ft_in_str:='';

mod_INCHES:= OSCAT_BASIC.MODR(inches_in,12);
div_FEET  := TO_REAL(FLOOR(inches_in/12.0));

Total_Inches:= (div_FEET * 12) + mod_INCHES;

IF div_FEET >= 1.0 THEN
	temp_ft_in_str := print_formated_REAl_func('',feet_format,div_FEET);
END_IF

temp_ft_in_str := CONCAT(temp_ft_in_str,print_formated_REAl_func(' ',inches_format,mod_INCHES));

Str:=temp_ft_in_str;
Inches:=mod_INCHES;
Feet:=TO_INT(div_FEET);

END_FUNCTION_BLOCK

// Device/Application/LIBS/Override_Timed
FUNCTION_BLOCK Override_Timed
VAR_INPUT
	ALLOW_IN: BOOL;
	ENABLE: BOOL;
	ALLOW_TIME:TIME;
END_VAR
VAR_OUTPUT
	ALLOW:BOOL;
	StatusString:STRING;
END_VAR
VAR
	ALLOW_TON: TON;
	RemainStr: STRING;
END_VAR

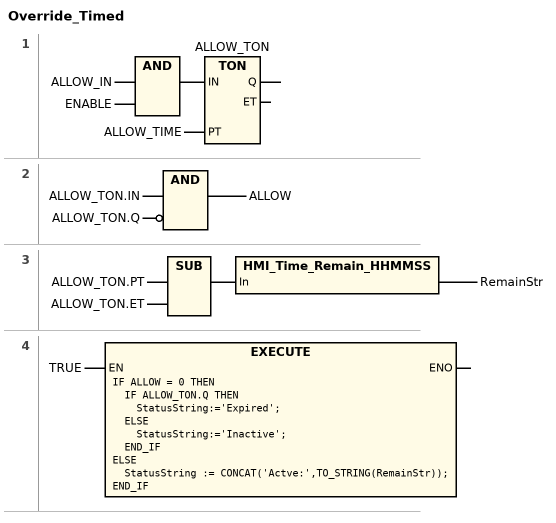
// NETWORK 1
ALLOW_TON(IN := ALLOW_IN AND ENABLE, PT := ALLOW_TIME); // TON

// NETWORK 2
ALLOW := ALLOW_TON.IN AND NOT ALLOW_TON.Q;

// NETWORK 3
RemainStr := HMI_Time_Remain_HHMMSS(In := ALLOW_TON.PT - ALLOW_TON.ET);

// NETWORK 4
IF ALLOW = 0 THEN
	IF ALLOW_TON.Q THEN
		StatusString:='Expired';		
	ELSE
		StatusString:='Inactive';		
	END_IF
ELSE
	StatusString := CONCAT('Actve:',TO_STRING(RemainStr));
END_IF

END_FUNCTION_BLOCK

// Device/Application/App_Common/Nav/Page Control/MoveArrow_1
FUNCTION_BLOCK MoveArrow_1
VAR_INPUT
	Enable: BOOL;
	LengthPoint: INT;
END_VAR
VAR_OUTPUT
	Out: INT;
	Invisible: BOOL;
END_VAR
VAR
	Ton1: TON;
	Count: INT;
END_VAR

Ton1(IN:= Enable AND NOT Ton1.Q, PT:=T#100MS);
IF Ton1.Q THEN
	Count:= Count + 5;
END_IF
IF Count>LengthPoint THEN Count:=0; END_IF
Out:=Count;
Invisible:= NOT Enable;

END_FUNCTION_BLOCK

// Device/Application/App_Common/Nav/Page Control/MoveArrow_2
FUNCTION_BLOCK MoveArrow_2
VAR_INPUT
	Enable: BOOL;
	LengthPoint: INT;
END_VAR
VAR_OUTPUT
	OutX: INT;
	OutY: INT;
	Invisible: BOOL;
END_VAR
VAR
	Ton1: TON;
	Count: INT;
	Count2: INT;

END_VAR

Ton1(IN:= Enable AND NOT Ton1.Q, PT:=T#100MS);
IF Ton1.Q THEN
	Count:= Count + 5;
	Count2:=REAL_TO_INT(0-(Count/2.222));
END_IF
IF Count>LengthPoint THEN Count:=0; Count2:=0; END_IF
OutX:=Count;
OutY:=Count2;
Invisible:= NOT Enable;

END_FUNCTION_BLOCK

// Device/Application/App_Common/Vizualisations/DIAG_IO/CR0403/CR0403_Output_Display
FUNCTION_BLOCK CR0403_Output_Display
VAR_INPUT
END_VAR
VAR_OUTPUT
	oPinDetailsStr:STRING;
	oSignalNameStr: STRING;
	oMainString: STRING; // could be Digital:ON/OFF, mV, mA or Hz PWM?
	oMainStringColour: DWORD;	
	oDiagStr: STRING; // Diagnostics info
	oShowDigRect:BOOL;
	oDigRectColour:DWORD;
	oTypeStr:STRING;
	oForceColour:DWORD;
	oForceText:STRING(5);
END_VAR
VAR
	InitDone:BOOL :=FALSE;	
	Update: BOOL:=TRUE;
	Update_Signal_Name: BOOL:=TRUE;	
	OpREF: REFERENCE TO OpCom_CR0403;
	Pin_Name_Temp:STRING(10);
	Pin_Number_Temp:STRING(10);
	temp_real_mA:STRING(10);
	temp_real_mV:STRING(10);
	TextListItem:STRING;
	MainStringFlash: BOOL;
	UpdateDiag: BOOL;
	MainStringTemp: STRING;
END_VAR

VAR_IN_OUT
END_VAR

IF Update=FALSE THEN
	RETURN;
END_IF

IF __ISVALIDREF(OpREF) = FALSE THEN
	RETURN;
END_IF

IF OpREF.RefsOK = FALSE THEN
	RETURN;
END_IF

// set defaults first for the main string
oShowDigRect:=FALSE;
oTypeStr:='';
MainStringFlash:=FALSE;
oMainString:='';
MainStringTemp:='';
oMainStringColour:=GVL_Viz.Diag_Output_Font_Colour_OK;
oTypeStr:='CSO-Hi';

// this code displays the Signal name - can be toggled using the function key
IF Update_Signal_Name THEN
	oPinDetailsStr:=OpREF.Pin_Name;
	IF GVL_Viz.Diag_Signal_Name_Toggle THEN
		TextListItem:=OpREF.Signal_Name;
	ELSE
		TextListItem:=Mimic_IO_GetText(GVL_Viz.TextList_IO_Diag,OpREF.PLC_IO_Ref);
	END_IF	
	
	IF (FIND(TextListItem,'Spare_') = 1) OR (FIND(TextListItem,'SPARE_') = 1) THEN
		// Starts with Spare
		oSignalNameStr:=' --- ';
	ELSE
		oSignalNameStr:=TextListItem;
	END_IF
END_IF

IF OpREF.Unavail THEN
	// the output is unvailable!
	IF GVL_Viz.Output_Fault_Flash_Slow THEN
		oMainString:=GVL_Viz.Diag_Output_Unavailable_Text;
		MainStringFlash:=TRUE;	
	END_IF
	oMainStringColour:=GVL_Viz.Diag_Output_Font_Colour_Unavail;
ELSIF OpREF.Diag_OK = FALSE THEN
	// something is not OK with the output
	// may be a fault or warning !
	IF GVL_Viz.Output_Fault_Flash_Slow THEN
		// do something if in this high period of the slow flash
		MainStringFlash:=TRUE;
		oMainString:=OpREF.DiagInfo;
	END_IF
	// always use the selected color - even if not showing the Diagnostic Info!
	IF OpREF.Diag_Error THEN
		oMainStringColour:=GVL_Viz.Diag_Output_Font_Colour_Error;
	ELSIF OpREF.Diag_Warn THEN
		oMainStringColour:=GVL_Viz.Diag_Output_Font_Colour_Warn;
	ELSE
		oMainStringColour:=GVL_Viz.Diag_Output_Font_Colour_Other;			
	END_IF			
END_IF


IF OpREF.Unavail=FALSE THEN
	// the output is unvailable!
	oShowDigRect:=TRUE;	
	UpdateDiag:=TRUE;
		
	IF OpREF.ValueFinalBool = FALSE THEN
		oDigRectColour:=GVL_Viz.IFM_IO_Output_DigRectColour_OFF;
		MainStringTemp:= CONCAT(MainStringTemp,'OFF');
	ELSE
		oDigRectColour:=GVL_Viz.IFM_IO_Output_DigRectColour_ON;
		MainStringTemp:= CONCAT(MainStringTemp,'ON');
	END_IF
	
END_IF
	
IF MainStringFlash = FALSE THEN
	oMainString:=MainStringTemp;
END_IF

// add the optional diagnostic string - maybe scaling information 
IF 	UpdateDiag=TRUE THEN
	IF LEN(OpREF.DiagString) > 0 THEN
		IF LEN(oMainString) > 0 THEN
			oMainString:= CONCAT(oMainString,',');		
		END_IF
		oMainString:= CONCAT(oMainString,OpREF.DiagString);
	END_IF	
END_IF

// show a special colour and M is the output is being force on with PLC Manual.
IF OpREF.OUTPUT_STATE_DATA.xManAuto THEN
	oForceText:='M';
	IF OpREF.OUTPUT_STATE_DATA.uiManValue > 0 THEN
		oForceColour:=GVL_Viz.IFM_IO_Output_DigRectColour_ManOn;
	ELSE
		oForceColour:=GVL_Viz.IFM_IO_Output_DigRectColour_ManOff;
	END_IF
ELSE
	oForceText:='';
	oForceColour:=16#FFFFFFFF;
END_IF

METHOD Init : BOOL
VAR_INPUT
	pOpREF: REFERENCE TO OpCom_CR0403;
END_VAR
OpREF REF= pOpREF;
InitDone:=TRUE;
END_METHOD

END_FUNCTION_BLOCK

// Device/Application/App_Common/Vizualisations/DIAG_IO/CR0403/OpCom_CR0403
FUNCTION_BLOCK OpCom_CR0403

VAR_INPUT
	Dig: BOOL;
	DiagString: STRING:='';	
END_VAR

VAR
	OUTPUT_STATE_DATA:  REFERENCE TO CRXXXX_OUTPUT_STATE_DATA;
	
	SET_UPDATES: DWORD;	
	PLC_Name: STRING;
	Signal_Name: STRING;
	Pin_Name: STRING;
	Pin_Details: STRING;
	
	NodeFB: REFERENCE TO NodeComFB;
	
	RefsOK: BOOL;
	
	Diag_OK:BOOL:=TRUE;
	Diag_Error:BOOL;
	Diag_Warn:BOOL;
	Diag_Other:BOOL;
	
	Fault:BOOL;	
	Unavail:BOOL;
	GroupSupplyOn:BOOL;
	
	DiagInfo:STRING:='';	
	PLC_IO_Ref:STRING;	
	
	Alarm_eDiagInfo:ifmTypes.DIAG_INFO;	
	AlmLog: IO_LogCom;
	Alarm_Active: BOOL;
END_VAR

VAR_OUTPUT
	ValueFinal: UINT;
	ValueFinalBool: BOOL;		
END_VAR

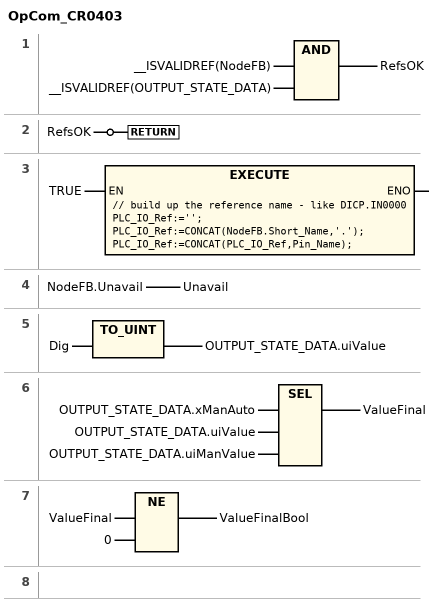
// NETWORK 1
RefsOK := (__ISVALIDREF(NodeFB)) AND (__ISVALIDREF(OUTPUT_STATE_DATA));

// NETWORK 2
IF NOT RefsOK THEN RETURN; END_IF

// NETWORK 3
// build up the reference name - like DICP.IN0000
PLC_IO_Ref:='';
PLC_IO_Ref:=CONCAT(NodeFB.Short_Name,'.');
PLC_IO_Ref:=CONCAT(PLC_IO_Ref,Pin_Name);

// NETWORK 4
Unavail := NodeFB.Unavail;

// NETWORK 5
OUTPUT_STATE_DATA.uiValue := TO_UINT(Dig);

// NETWORK 6
ValueFinal := SEL(OUTPUT_STATE_DATA.xManAuto, OUTPUT_STATE_DATA.uiValue, OUTPUT_STATE_DATA.uiManValue);

// NETWORK 7
ValueFinalBool := ValueFinal <> 0;

// NETWORK 8

PROPERTY uValue : UINT
GET
IF __ISVALIDREF(OUTPUT_STATE_DATA) THEN
	uValue:=OUTPUT_STATE_DATA.uiValue;
END_IF
END_GET
SET
IF __ISVALIDREF(OUTPUT_STATE_DATA) THEN
	OUTPUT_STATE_DATA.uiValue:=uValue;
END_IF
END_SET
END_PROPERTY

METHOD Init : BOOL
VAR_INPUT
	pPLC_Name: STRING;
	pSignal_Name: STRING;
	pPin_Name: STRING;
	pPin_Details: STRING;
	pOUTPUT_STATE_DATA: REFERENCE TO CRXXXX_OUTPUT_STATE_DATA;	
	pNodeFB: REFERENCE TO NodeComFB;
END_VAR

PLC_Name:=pPLC_Name;
Signal_Name:=pSignal_Name;
Pin_Name:=pPin_Name;
Pin_Details:=pPin_Details;

OUTPUT_STATE_DATA REF= pOUTPUT_STATE_DATA;

NodeFB REF=pNodeFB;
END_METHOD

END_FUNCTION_BLOCK

// Device/Application/App_Common/Vizualisations/Main/Visualization_Settings_Main
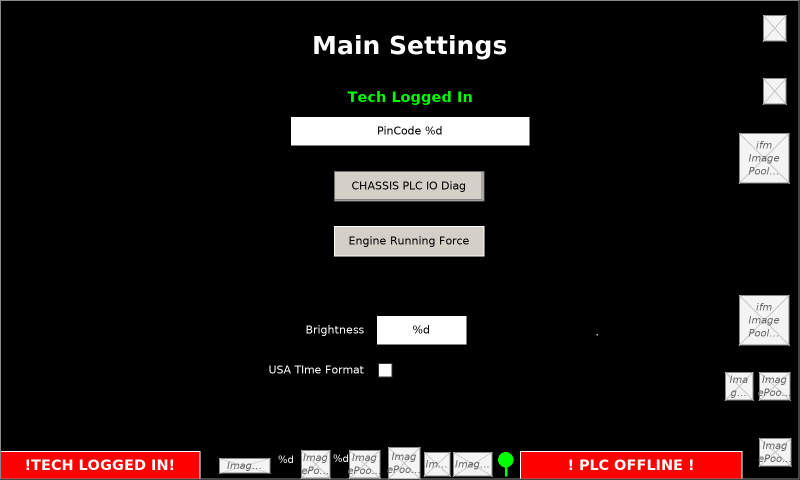
VISUALIZATION Visualization_Settings_Main  // 800x480
    Frame (0,0 800x480)
        shows Visualization_Template()
    Button (334,171 150x30), "CHASSIS PLC IO Diag"
        tap Nav.NAV_TO_IO_DIAG_PAGES
    Label (219,30 382x30), "Main Settings"
    Rectangle (290,116 240x30), "PinCode %d", text variable: SECURITY_COM.PIN_CODE_ENTERED
        OnMouseClick: write the text variable via VisuDialogs_Template.Numpad, min 0, max 9999, title '4 digit pincode'
    Label (327,86 167x22), "Tech Logged In", invisible if: NOT GVL_System.Access_Level_Tech
    Image (739,295 50x50), image: ifmImagePool.Engine Icon50pixel
    Image (759,372 31x28), image: ImagePool.Hazard_31_28
    Image (725,372 28x28), image: ImagePool.warning_28_28
    Image (597,334 0x1), image: ImagePool.settings
    Rectangle (376,315 91x30), "%d", text variable: GVL_Persistant.Brightness
        OnValueChanged: execute {  }
        OnValueChanged: write the text variable via Default, min LCD_Brighness_Control.Brightness_Min, max LCD_Brighness_Control.Brightness_Max
        OnMouseClick: write the text variable via VisuDialogs_Template.Numpad, min 10, max 100, title 'Brighntess %'
    Label (291,315 76x30), "Brightness"
    Image (739,133 50x50), image: ifmImagePool.speedometer50pixel
    Image (763,15 23x26), invisible if: Nav.Footer_ShowNavLeft=0, image: ImagePool.Page_nav_left
    Image (763,78 23x26), invisible if: Nav.Footer_ShowNavRight=0, image: ImagePool.Page_nav_right
    Rectangle (334,226 150x30), "Engine Running Force", invisible if: GVL_System.Access_Level_Tech=0, input disabled if: GVL_System.Access_Level_Tech=0
        toggle GVL_Machine.EngineRunningForce
    Checkbox (376,355 33x30), variable: GVL_Persistant.Sys_Settings.USA_TIme_Format
    Label (251,355 116x30), "USA TIme Format"
END_VISUALIZATION

// Device/Application/App_Common/Vizualisations/Main/Layout/Visualization_Footer
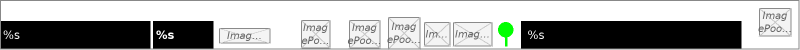
VISUALIZATION Visualization_Footer  // 800x50
    Image (301,20 28x28), image: ImagePool.warning_28_28_dull
    Image (349,20 31x28), image: ImagePool.Hazard_31_28_dull
    Image (759,8 32x28), image: ImagePool.home
    Image (388,17 32x32), image: ImagePool.settings
    Image (349,20 31x28), invisible if: NVL_Viz.Sections.Footer.ShowErrorIcon=0, image: ImagePool.Hazard_31_28
    Image (301,20 29x28), invisible if: NVL_Viz.Sections.Footer.ShowWarningIcon=0, image: ImagePool.warning_28_28
    Rectangle (269,21 28x17), "%d", text variable: NVL_Viz.Sections.Footer.NumberWarnings, invisible if: NVL_Viz.Sections.Footer.NumberWarnings=0
    Rectangle (324,20 28x17), "%d", text variable: NVL_Viz.Sections.Footer.NumberErrors, invisible if: NVL_Viz.Sections.Footer.NumberErrors=0
    Image (388,17 32x32), invisible if: NOT GVL_System.Access_Level_Tech, image: ImagePool.settings_32_32_green
    Rectangle (521,21 220x28), "%s", text variable: NVL_Viz.Sections.Footer.Header_Message_Str, invisible if: NOT NVL_Viz.Sections.Footer.Header_Message_Show_Flash
        p55702900: NVL_Viz.Sections.Footer.Header_Message_Colour
    Rectangle (521,21 220x28), "%s", text variable: NVL_Viz.Sections.Footer.DisplayDateTimeString, invisible if: NVL_Viz.Sections.Footer.Header_Message_Show_RTC=0
    Rectangle (0,21 150x28), "%s", text variable: Nav.Head_PageName
    Image (424,22 26x24), invisible if: NOT NVL_Viz.Sections.Footer.Siren, image: ImagePool.Header_Siren
    Image (453,22 39x24), invisible if: NOT NVL_Viz.Sections.Footer.Beacon, image: ImagePool.Header_Beacon
    Line (951,260)
    Image (219,28 51x15), invisible if: GVL_Machine.TrackingModeAllow=0, image: ImagePool.Tracks_51_15_white
    Image (219,28 51x15), invisible if: GVL_Machine.TrackingMode=0 AND GVL_Machine.TrackPreSiren_Flash=0, image: ImagePool.Tracks_51_15_orange
    Rectangle (153,21 60x28), "%s", text variable: NVL_Viz.Sections.Footer.SystemVoltageStr, invisible if: NOT NVL_Viz.Sections.Footer.SystemVoltageVisable
        p55702900: NVL_Viz.Sections.Footer.SystemVoltageColour
    Ellipse (498,22 15x15), invisible if: GVL_Machine.SetupDumpValveIcon=0
    Rectangle (505,36 2x10), invisible if: GVL_Machine.SetupDumpValveIcon=0
END_VISUALIZATION

// Device/Application/App_Common/Vizualisations/Main/Layout/Visualization_Keypad_PC_SIM
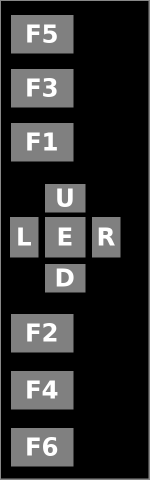
VISUALIZATION Visualization_Keypad_PC_SIM  // 150x480
    Rectangle (0,0 150x480)
    Rectangle (10,14 64x40), "F5"
        tap GVL_KeyList.xF5
    Rectangle (10,68 64x40), "F3"
        tap GVL_KeyList.xF3
    Rectangle (10,122 64x40), "F1"
        tap GVL_KeyList.xF1
    Rectangle (10,313 64x40), "F2"
        tap GVL_KeyList.xF2
    Rectangle (10,370 64x40), "F4"
        tap GVL_KeyList.xF4
    Rectangle (10,427 64x40), "F6"
        tap GVL_KeyList.xF6
    Rectangle (91,216 30x42), "R"
        tap GVL_KeyList.xRight
    Rectangle (44,263 42x30), "D"
        tap GVL_KeyList.xDown
    Rectangle (44,216 42x42), "E"
        tap GVL_KeyList.xKey_Return
    Rectangle (9,216 30x42), "L"
        tap GVL_KeyList.xLeft
    Rectangle (44,183 42x30), "U"
        tap GVL_KeyList.xUp
END_VISUALIZATION

// Device/Application/App_Common/Vizualisations/Main/Visualization_Alarms_Main
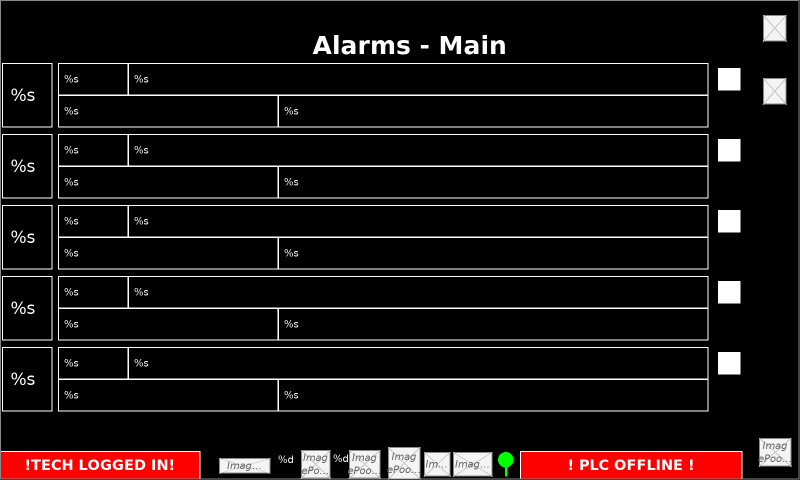
VISUALIZATION Visualization_Alarms_Main  // 800x480
VAR_IN_OUT
END_VAR
VAR
	bFreezeScrlPos : BOOL;
END_VAR
    Frame (0,0 800x480)
        shows Visualization_Template()
    Label (219,30 382x30), "Alarms - Main"
    Frame (0,62 707x348)
        shows Alarm_Logger_Table(LINE := Alarm_Table_Main.Lines)
    Image (763,15 23x26), invisible if: Nav.Footer_ShowNavLeft=0, image: ImagePool.Page_nav_left
    Image (763,78 23x26), invisible if: Nav.Footer_ShowNavRight=0, image: ImagePool.Page_nav_right
END_VISUALIZATION

// Device/Application/App_Common/Vizualisations/DIAG_IO/Visualization_DIAG_IO_Op_G0
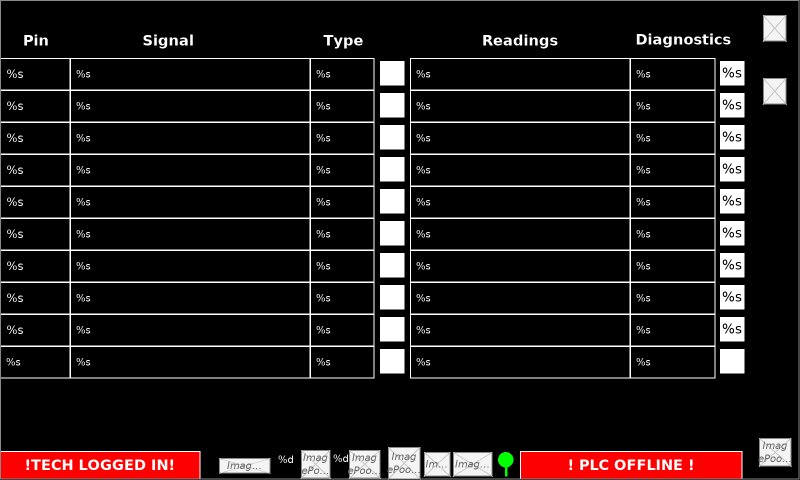
VISUALIZATION Visualization_DIAG_IO_Op_G0  // 800x480
    Frame (0,0 800x480)
        shows Visualization_Template()
    Frame (0,25 800x424)
        shows Visualization_CR0709_Op_G0(HMI_PLC_IO := HMI_IO.CHASSIS)
    Image (763,15 23x26), invisible if: Nav.Footer_ShowNavLeft=0, image: ImagePool.Page_nav_left
    Image (763,78 23x26), invisible if: Nav.Footer_ShowNavRight=0, image: ImagePool.Page_nav_right
END_VISUALIZATION

// Device/Application/App_Common/Vizualisations/Main/Layout/Visualization_Template
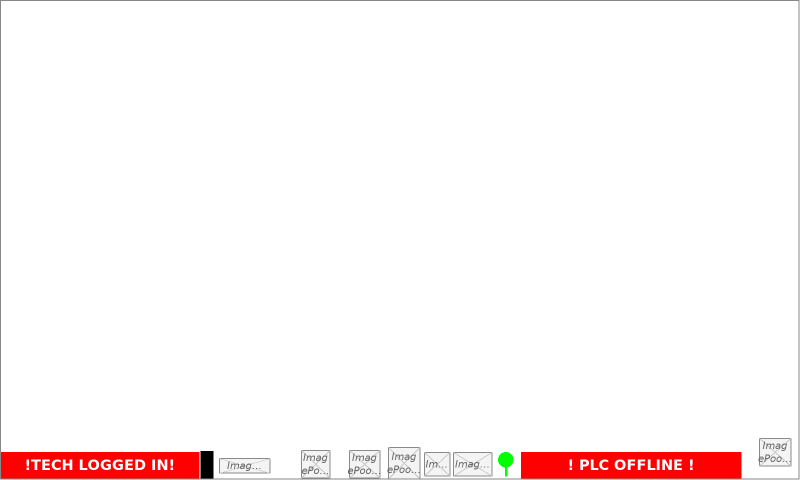
VISUALIZATION Visualization_Template  // 800x480
    Frame (0,430 800x50), frame switch variable: PLC_COMMON.PC_SIMULATION_MODE
        shows Visualization_Footer()
        shows Visualization_Footer_PC_SIM()
    TabControl (958,0 700x750), invisible if: PLC_COMMON.PC_SIMULATION_MODE=0, input disabled if: PLC_COMMON.PC_SIMULATION_MODE=0, frame switch variable: GVL_System.SIM_IO_TAB_INDEX
        shows Visualization_SIM_IO()
        shows Visualization_SIM_IO_AUX()
        shows Visualization_SIM_IO_CAS()
        [0]: TabTitle=Main
        [1]: TabTitle=Aux
    Frame (800,0 150x480), invisible if: PLC_COMMON.PC_SIMULATION_MODE=0, input disabled if: PLC_COMMON.PC_SIMULATION_MODE=0
        shows Visualization_Keypad_PC_SIM()
    RoundedRectangle (520,451 222x28), "! PLC OFFLINE !", invisible if: Machine_IO.Node_CHASSIS.Unavail=0 OR GVL_Viz.Common_Flash_Fast=0
    RoundedRectangle (0,451 200x28), "!TECH LOGGED IN!", invisible if: GVL_System.Access_Level_Tech=0 OR GVL_Viz.Common_Flash_Fast=0
END_VISUALIZATION

// Device/Application/App_Common/Vizualisations/Main/Visualization_PLC_Versions
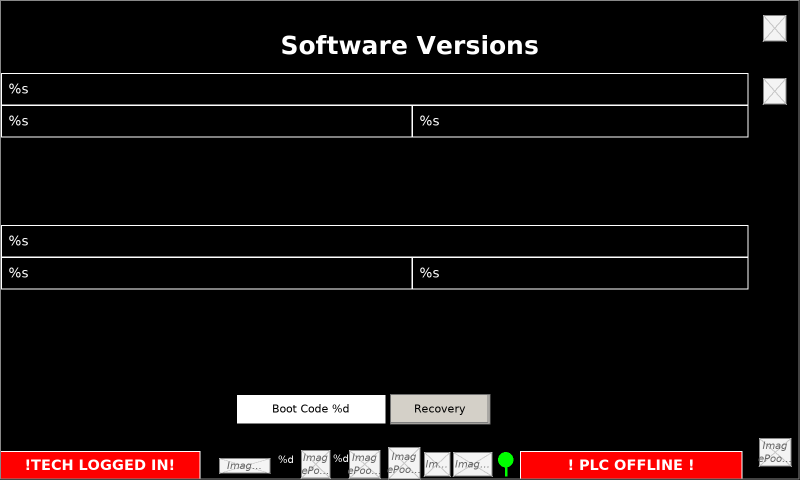
VISUALIZATION Visualization_PLC_Versions  // 800x480
    Frame (0,0 800x480)
        shows Visualization_Template()
    Label (219,30 382x30), "Software Versions"
    Frame (0,225 800x50)
        shows PLC_Version_Info(PlcVersion := PLC_COMMON.CHASSIS_PLC_Version_Info)
    Frame (0,73 800x50)
        shows PLC_Version_Info(PlcVersion := PLC_COMMON.MAIN_HMI_Version_Info)
    Rectangle (236,394 150x30), "Boot Code %d", text variable: PLC_COMMON.BOOT_PIN_CODE_ENTERED
        OnMouseClick: write the text variable via Default, min 0, max 9999, title 'Boot 4 digit pincode'
    Button (390,394 100x30), "Recovery", invisible if: PLC_COMMON.BOOT_PIN_CODE_VALID=0
        tap PLC_COMMON.BOOT_INTO_RECOVERY
    Image (763,15 23x26), invisible if: Nav.Footer_ShowNavLeft=0, image: ImagePool.Page_nav_left
    Image (763,78 23x26), invisible if: Nav.Footer_ShowNavRight=0, image: ImagePool.Page_nav_right
END_VISUALIZATION

// Device/Application/LIBS/IO Diagnostics/IO Page Templates/CR0709/Visualization_CR0709_Op_G1
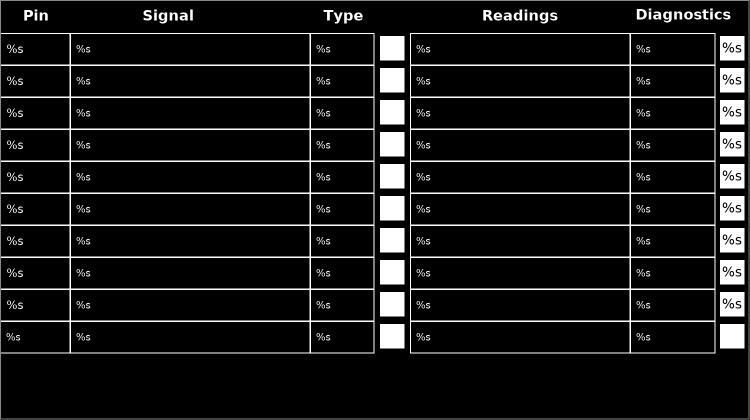
VISUALIZATION Visualization_CR0709_Op_G1  // 750x420
VAR_IN_OUT
	HMI_PLC_IO: HMI_PLC_CR0709_IO;
END_VAR
    Frame (0,33 762x32)
        shows Output_IFM_PLC_CRXXXX(Output := HMI_PLC_IO.OUT0100)
    Frame (0,0 750x32)
        shows Output_IFM_PLC_CRXXXX_TITLE()
    Frame (0,65 762x32)
        shows Output_IFM_PLC_CRXXXX(Output := HMI_PLC_IO.OUT0101)
    Frame (0,97 762x32)
        shows Output_IFM_PLC_CRXXXX(Output := HMI_PLC_IO.OUT0102)
    Frame (0,129 762x32)
        shows Output_IFM_PLC_CRXXXX(Output := HMI_PLC_IO.OUT0103)
    Frame (0,161 762x32)
        shows Output_IFM_PLC_CRXXXX(Output := HMI_PLC_IO.OUT0104)
    Frame (0,193 762x32)
        shows Output_IFM_PLC_CRXXXX(Output := HMI_PLC_IO.OUT0105)
    Frame (0,225 762x32)
        shows Output_IFM_PLC_CRXXXX(Output := HMI_PLC_IO.OUT0106)
    Frame (0,257 762x32)
        shows Output_IFM_PLC_CRXXXX(Output := HMI_PLC_IO.OUT0107)
    Frame (0,289 762x32)
        shows Output_IFM_PLC_CRXXXX(Output := HMI_PLC_IO.OUT0108)
    Frame (0,321 780x32)
        shows Output_Group_IFM_PLC_CRXXXX(Output := HMI_PLC_IO.GROUP1)
END_VISUALIZATION

// Device/Application/App_Common/Vizualisations/DIAG_IO/Visualization_DIAG_IO_Ip_G1
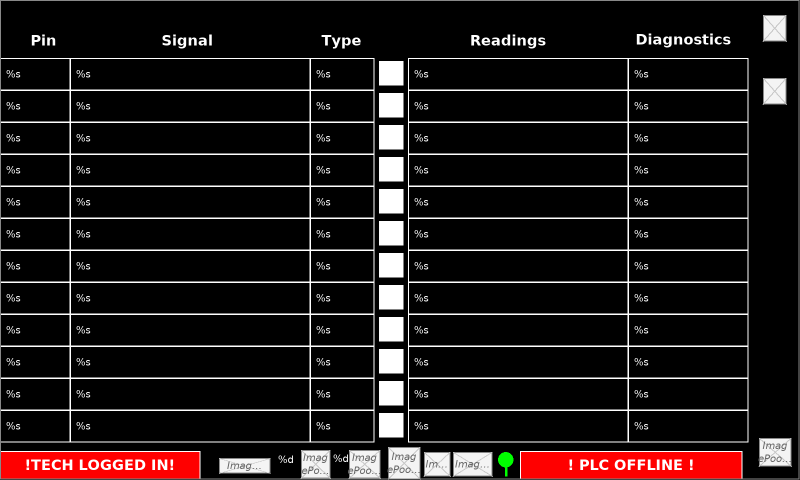
VISUALIZATION Visualization_DIAG_IO_Ip_G1  // 800x480
    Frame (0,0 800x480)
        shows Visualization_Template()
    Frame (0,25 800x424)
        shows Visualization_CR0709_Ip_G1(HMI_PLC_IO := HMI_IO.CHASSIS)
    Image (763,15 23x26), invisible if: Nav.Footer_ShowNavLeft=0, image: ImagePool.Page_nav_left
    Image (763,78 23x26), invisible if: Nav.Footer_ShowNavRight=0, image: ImagePool.Page_nav_right
END_VISUALIZATION

// Device/Application/App_Common/Vizualisations/DIAG_IO/Visualization_DIAG_IO_Ip_G2
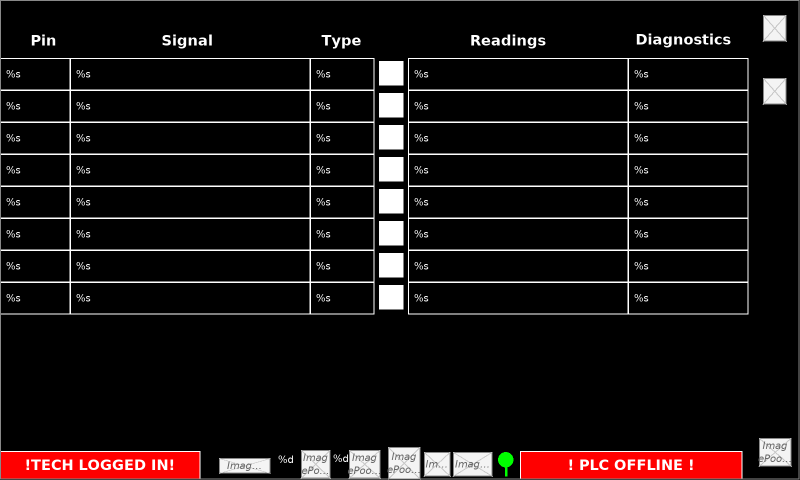
VISUALIZATION Visualization_DIAG_IO_Ip_G2  // 800x480
    Frame (0,0 800x480)
        shows Visualization_Template()
    Frame (0,25 800x424)
        shows Visualization_CR0709_Ip_G2(HMI_PLC_IO := HMI_IO.CHASSIS)
    Image (763,15 23x26), invisible if: Nav.Footer_ShowNavLeft=0, image: ImagePool.Page_nav_left
    Image (763,78 23x26), invisible if: Nav.Footer_ShowNavRight=0, image: ImagePool.Page_nav_right
END_VISUALIZATION

// Device/Application/App_Common/Vizualisations/DIAG_IO/Visualization_DIAG_IO_Op_G1
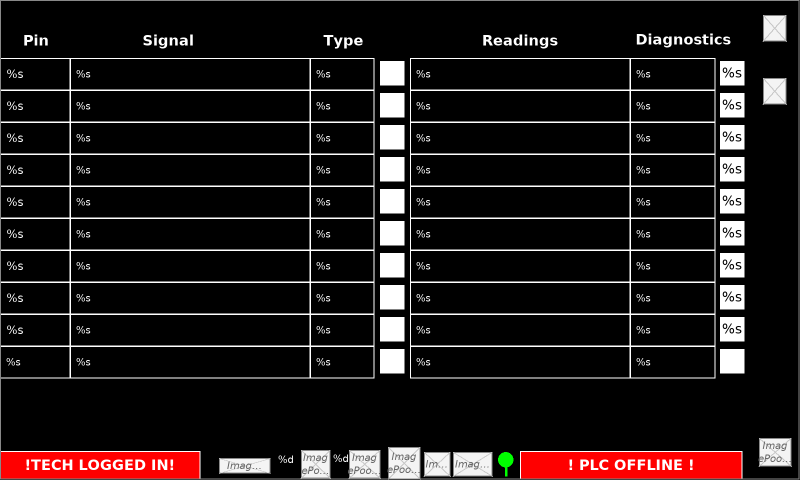
VISUALIZATION Visualization_DIAG_IO_Op_G1  // 800x480
    Frame (0,0 800x480)
        shows Visualization_Template()
    Frame (0,25 800x424)
        shows Visualization_CR0709_Op_G1(HMI_PLC_IO := HMI_IO.CHASSIS)
    Image (763,15 23x26), invisible if: Nav.Footer_ShowNavLeft=0, image: ImagePool.Page_nav_left
    Image (763,78 23x26), invisible if: Nav.Footer_ShowNavRight=0, image: ImagePool.Page_nav_right
END_VISUALIZATION

// Device/Application/App_Common/Vizualisations/DIAG_IO/Visualization_DIAG_IO_Op_G2
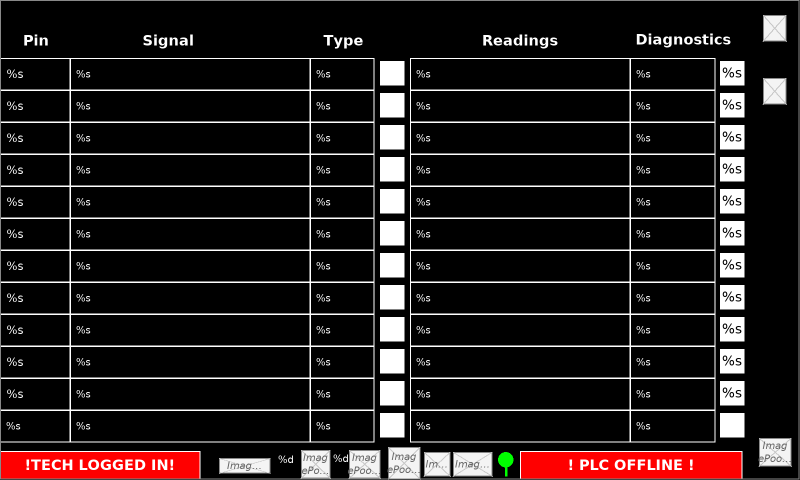
VISUALIZATION Visualization_DIAG_IO_Op_G2  // 800x480
    Frame (0,0 800x480)
        shows Visualization_Template()
    Frame (0,25 800x424)
        shows Visualization_CR0709_Op_G2(HMI_PLC_IO := HMI_IO.CHASSIS)
    Image (763,15 23x26), invisible if: Nav.Footer_ShowNavLeft=0, image: ImagePool.Page_nav_left
    Image (763,78 23x26), invisible if: Nav.Footer_ShowNavRight=0, image: ImagePool.Page_nav_right
END_VISUALIZATION

// Device/Application/App_Common/Vizualisations/DIAG_IO/Visualization_DIAG_IO_Ip_G0
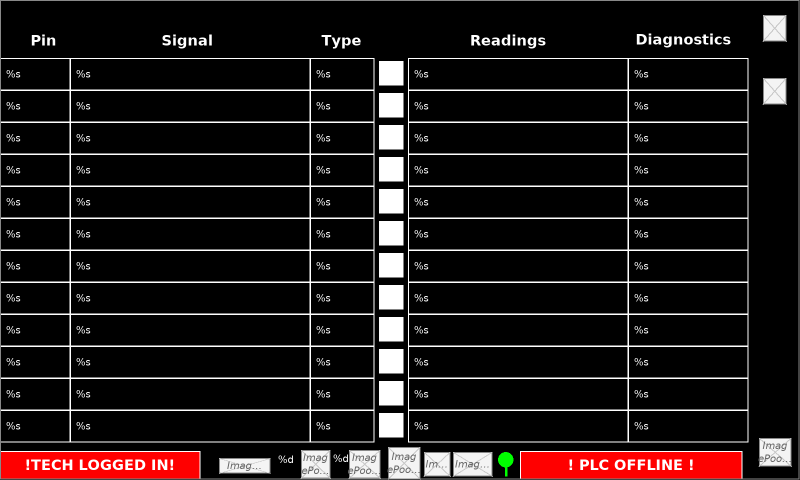
VISUALIZATION Visualization_DIAG_IO_Ip_G0  // 800x480
    Frame (0,0 800x480)
        shows Visualization_Template()
    Frame (0,25 800x424)
        shows Visualization_CR0709_Ip_G0(HMI_PLC_IO := HMI_IO.CHASSIS)
    Image (763,15 23x26), invisible if: Nav.Footer_ShowNavLeft=0, image: ImagePool.Page_nav_left
    Image (763,78 23x26), invisible if: Nav.Footer_ShowNavRight=0, image: ImagePool.Page_nav_right
END_VISUALIZATION

// Device/Application/LIBS/IO Diagnostics/IO Page Templates/CR0709/Visualization_CR0709_Ip_G2
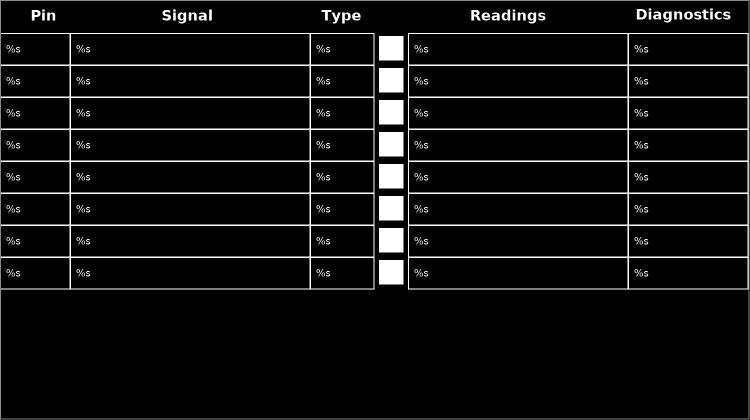
VISUALIZATION Visualization_CR0709_Ip_G2  // 750x420
VAR_IN_OUT
	HMI_PLC_IO: HMI_PLC_CR0709_IO;
END_VAR
    Frame (0,33 762x32)
        shows Input_IFM_PLC_CRXXXX(Input := HMI_PLC_IO.IN0400)
    Frame (0,0 801x32)
        shows Input_IFM_PLC_CRXXXX_TITLE()
    Frame (0,65 762x32)
        shows Input_IFM_PLC_CRXXXX(Input := HMI_PLC_IO.IN0401)
    Frame (0,97 762x32)
        shows Input_IFM_PLC_CRXXXX(Input := HMI_PLC_IO.IN0900)
    Frame (0,129 762x32)
        shows Input_IFM_PLC_CRXXXX(Input := HMI_PLC_IO.IN0901)
    Frame (0,161 762x32)
        shows Input_IFM_PLC_CRXXXX(Input := HMI_PLC_IO.IN0300)
    Frame (0,193 762x32)
        shows Input_IFM_PLC_CRXXXX(Input := HMI_PLC_IO.IN0301)
    Frame (0,225 762x32)
        shows Input_IFM_PLC_CRXXXX(Input := HMI_PLC_IO.IN0800)
    Frame (0,257 762x32)
        shows Input_IFM_PLC_CRXXXX(Input := HMI_PLC_IO.IN0801)
END_VISUALIZATION

// Device/Application/LIBS/IO Diagnostics/IO Page Templates/UDP/PLC_UDP_Info
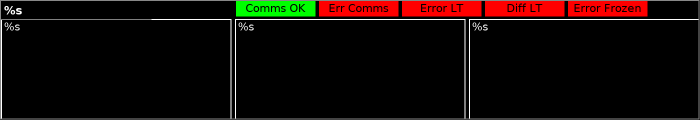
VISUALIZATION PLC_UDP_Info  // 700x120
VAR_IN_OUT
	UDP_Info: UDP_Info_Viz;
END_VAR
    Textfield (1,19 230x100), "%s", text variable: UDP_Info.InfoString
    Textfield (235,19 230x100), "%s", text variable: UDP_Info.ErrString
    Textfield (469,19 230x100), "%s", text variable: UDP_Info.WarnString
    Rectangle (568,1 79x15), "Error Frozen", invisible if: NOT UDP_Info.Frozen_Error
    Rectangle (485,1 79x15), "Diff LT", invisible if: NOT UDP_Info.Diff_Error
    Rectangle (402,1 79x15), "Error LT", invisible if: NOT UDP_Info.LT_Error
    Rectangle (319,1 79x15), "Err Comms", invisible if: NOT UDP_Info.CommsError
    Rectangle (236,1 79x15), "Comms OK", invisible if: UDP_Info.CommsError
    Rectangle (1,2 150x17), "%s", text variable: UDP_Info.NodeName
END_VISUALIZATION

// Device/Application/LIBS/IO Diagnostics/IO Page Templates/PLC_Status/PLC_Status_Info
